C09277=1102.667,-32.003,-50.837,179.868,5.922,149.097
C09278=1102.672,-32.217,-50.825,179.868,5.919,149.097
C09279=1102.676,-32.431,-50.814,179.868,5.915,149.096
C09280=1102.682,-32.681,-50.801,179.867,5.910,149.095
C09281=1102.687,-32.930,-50.787,179.867,5.906,149.094
C09282=1102.692,-33.180,-50.774,179.867,5.902,149.093
C09283=1102.697,-33.429,-50.761,179.866,5.897,149.092
C09284=1102.702,-33.679,-50.748,179.866,5.893,149.091
C09285=1102.707,-33.928,-50.734,179.866,5.889,149.090
C09286=1102.712,-34.178,-50.721,179.865,5.884,149.089
C09287=1102.717,-34.428,-50.708,179.865,5.879,149.089
C09288=1102.723,-34.677,-50.696,179.865,5.875,149.088
C09289=1102.727,-34.927,-50.683,179.865,5.870,149.087
C09290=1102.733,-35.176,-50.669,179.864,5.866,149.086
C09291=1102.737,-35.426,-50.656,179.864,5.862,149.085
C09292=1102.743,-35.676,-50.643,179.864,5.857,149.084
C09293=1102.748,-35.926,-50.630,179.863,5.852,149.083
C09294=1102.753,-36.175,-50.617,179.864,5.848,149.082
C09295=1102.758,-36.424,-50.603,179.863,5.844,149.081
C09296=1102.763,-36.674,-50.590,179.863,5.839,149.080
C09297=1102.768,-36.924,-50.577,179.863,5.835,149.079
C09298=1102.774,-37.173,-50.564,179.862,5.830,149.079
C09299=1102.778,-37.423,-50.551,179.862,5.826,149.078
C09300=1102.783,-37.673,-50.539,179.862,5.822,149.077
C09301=1102.789,-37.923,-50.525,179.862,5.817,149.076
C09302=1102.794,-38.172,-50.513,179.861,5.812,149.075
C09303=1102.799,-38.421,-50.499,179.861,5.807,149.074
C09304=1102.804,-38.671,-50.486,179.861,5.803,149.073
C09305=1102.809,-38.921,-50.473,179.861,5.798,149.072
C09306=1102.814,-39.170,-50.460,179.860,5.794,149.071
C09307=1102.819,-39.420,-50.447,179.861,5.790,149.070
C09308=1102.825,-39.670,-50.434,179.860,5.785,149.069
C09309=1102.830,-39.919,-50.422,179.860,5.780,149.068
C09310=1102.834,-40.169,-50.409,179.860,5.775,149.067
C09311=1102.840,-40.419,-50.396,179.860,5.771,149.066
C09312=1102.845,-40.668,-50.383,179.860,5.766,149.065
C09313=1102.850,-40.918,-50.370,179.860,5.761,149.064
C09314=1102.855,-41.167,-50.357,179.860,5.757,149.063
C09315=1102.861,-41.417,-50.344,179.860,5.752,149.062
C09316=1102.865,-41.667,-50.331,179.859,5.748,149.061
C09317=1102.870,-41.916,-50.319,179.859,5.742,149.060
C09318=1102.875,-42.166,-50.306,179.859,5.738,149.059
C09319=1102.881,-42.415,-50.293,179.860,5.733,149.058
C09320=1102.886,-42.665,-50.280,179.859,5.729,149.057
C09321=1102.891,-42.915,-50.267,179.859,5.723,149.056
C09322=1102.896,-43.164,-50.255,179.860,5.719,149.055
C09323=1102.901,-43.414,-50.242,179.860,5.714,149.054
C09324=1102.906,-43.663,-50.228,179.859,5.709,149.053
C09325=1102.912,-43.913,-50.217,179.860,5.705,149.052
C09326=1102.916,-44.163,-50.204,179.860,5.700,149.050
C09327=1102.922,-44.413,-50.191,179.860,5.695,149.049
C09328=1102.926,-44.627,-50.180,179.860,5.691,149.048
C09329=1102.931,-44.841,-50.169,179.861,5.687,149.047
C09330=1102.935,-45.055,-50.159,179.861,5.683,149.046
C09331=1102.939,-45.269,-50.147,179.861,5.679,149.046
C09332=1102.943,-45.483,-50.136,179.861,5.675,149.045
C09333=1102.947,-45.697,-50.125,179.861,5.671,149.044
C09334=1102.952,-45.911,-50.115,179.861,5.667,149.043
C09335=1102.957,-46.126,-50.103,179.862,5.663,149.042
C09336=1102.962,-46.375,-50.091,179.862,5.658,149.041
C09337=1102.967,-46.626,-50.079,179.862,5.653,149.040
C09338=1102.972,-46.875,-50.066,179.862,5.649,149.039
C09339=1102.977,-47.124,-50.053,179.862,5.644,149.037
C09340=1102.982,-47.373,-50.041,179.862,5.639,149.036
C09341=1102.987,-47.623,-50.028,179.862,5.635,149.035
C09342=1102.993,-47.874,-50.015,179.862,5.630,149.034
C09343=1102.998,-48.123,-50.003,179.862,5.625,149.033
C09344=1103.003,-48.372,-49.990,179.863,5.621,149.032
C09345=1103.008,-48.622,-49.978,179.863,5.616,149.031
C09346=1103.013,-48.872,-49.965,179.863,5.610,149.030
C09347=1103.018,-49.122,-49.953,179.863,5.606,149.029
C09348=1103.023,-49.371,-49.940,179.863,5.601,149.028
C09349=1103.028,-49.620,-49.928,179.863,5.596,149.027
C09350=1103.034,-49.870,-49.916,179.864,5.592,149.026
C09351=1103.039,-50.120,-49.903,179.863,5.587,149.025
C09352=1103.044,-50.370,-49.890,179.864,5.583,149.023
C09353=1103.049,-50.619,-49.877,179.864,5.578,149.022
C09354=1103.054,-50.869,-49.866,179.864,5.573,149.021
C09355=1103.059,-51.118,-49.853,179.864,5.569,149.020
C09356=1103.064,-51.367,-49.840,179.864,5.564,149.019
C09357=1103.070,-51.617,-49.829,179.864,5.559,149.018
C09358=1103.074,-51.867,-49.816,179.865,5.555,149.017
C09359=1103.079,-52.117,-49.803,179.865,5.549,149.016
C09360=1103.085,-52.367,-49.791,179.864,5.545,149.015
C09361=1103.090,-52.616,-49.778,179.865,5.540,149.014
C09362=1103.095,-52.865,-49.766,179.865,5.535,149.013
C09363=1103.101,-53.115,-49.754,179.865,5.530,149.012
C09364=1103.105,-53.365,-49.741,179.865,5.526,149.011
C09365=1103.110,-53.615,-49.729,179.865,5.521,149.009
C09366=1103.116,-53.864,-49.717,179.865,5.516,149.008
C09367=1103.121,-54.114,-49.704,179.866,5.512,149.007
C09368=1103.126,-54.364,-49.692,179.865,5.507,149.006
C09369=1103.131,-54.613,-49.679,179.865,5.502,149.005
C09370=1103.137,-54.863,-49.668,179.866,5.498,149.004
C09371=1103.142,-55.112,-49.655,179.866,5.493,149.003
C09372=1103.146,-55.362,-49.642,179.866,5.488,149.002
C09373=1103.152,-55.612,-49.630,179.866,5.484,149.001
C09374=1103.157,-55.862,-49.617,179.866,5.479,149.000
C09375=1103.162,-56.112,-49.606,179.866,5.474,148.999
C09376=1103.167,-56.361,-49.593,179.866,5.470,148.998
C09377=1103.172,-56.610,-49.582,179.866,5.465,148.997
C09378=1103.177,-56.860,-49.569,179.866,5.460,148.995
C09379=1103.183,-57.110,-49.557,179.867,5.456,148.995
C09380=1103.188,-57.359,-49.545,179.867,5.450,148.993
C09381=1103.193,-57.609,-49.533,179.866,5.446,148.992
C09382=1103.198,-57.859,-49.520,179.867,5.441,148.991
C09383=1103.203,-58.109,-49.508,179.867,5.436,148.990
C09384=1103.208,-58.322,-49.498,179.867,5.432,148.989
C09385=1103.212,-58.537,-49.487,179.867,5.429,148.989
C09386=1103.216,-58.752,-49.477,179.867,5.424,148.988
C09387=1103.221,-58.965,-49.466,179.867,5.420,148.987
C09388=1103.225,-59.179,-49.456,179.867,5.416,148.986
C09389=1103.229,-59.394,-49.446,179.867,5.412,148.985
C09390=1103.234,-59.608,-49.435,179.867,5.408,148.984
C09391=1103.238,-59.822,-49.425,179.868,5.404,148.983
C09392=1103.243,-60.072,-49.413,179.867,5.400,148.982
C09393=1103.249,-60.322,-49.401,179.867,5.394,148.981
C09394=1103.254,-60.571,-49.388,179.867,5.390,148.980
C09395=1103.259,-60.821,-49.376,179.867,5.385,148.979
C09396=1103.264,-61.070,-49.364,179.867,5.380,148.978
C09397=1103.269,-61.320,-49.353,179.866,5.375,148.977
C09398=1103.275,-61.570,-49.341,179.866,5.370,148.976
C09399=1103.280,-61.819,-49.328,179.866,5.365,148.975
C09400=1103.284,-62.069,-49.317,179.866,5.360,148.974
C09401=1103.290,-62.319,-49.305,179.866,5.355,148.973
C09402=1103.295,-62.568,-49.292,179.866,5.350,148.972
C09403=1103.300,-62.818,-49.280,179.866,5.345,148.970
C09404=1103.305,-63.068,-49.269,179.866,5.340,148.969
C09405=1103.310,-63.317,-49.256,179.866,5.335,148.968
C09406=1103.316,-63.567,-49.245,179.865,5.330,148.967
C09407=1103.321,-63.817,-49.233,179.865,5.325,148.966
C09408=1103.326,-64.067,-49.221,179.865,5.321,148.965
C09409=1103.331,-64.316,-49.209,179.865,5.315,148.964
C09410=1103.336,-64.566,-49.197,179.865,5.310,148.963
C09411=1103.341,-64.815,-49.186,179.865,5.306,148.962
C09412=1103.346,-65.065,-49.174,179.865,5.300,148.961
C09413=1103.351,-65.315,-49.161,179.865,5.295,148.960
C09414=1103.357,-65.565,-49.149,179.865,5.291,148.959
C09415=1103.362,-65.814,-49.138,179.865,5.285,148.958
C09416=1103.367,-66.064,-49.126,179.865,5.280,148.956
C09417=1103.372,-66.314,-49.113,179.865,5.276,148.956
C09418=1103.377,-66.563,-49.102,179.865,5.270,148.954
C09419=1103.382,-66.813,-49.090,179.865,5.265,148.953
C09420=1103.388,-67.062,-49.079,179.864,5.261,148.952
C09421=1103.393,-67.312,-49.068,179.865,5.255,148.951
C09422=1103.398,-67.562,-49.056,179.865,5.250,148.950
C09423=1103.403,-67.811,-49.044,179.865,5.245,148.949
C09424=1103.408,-68.061,-49.032,179.865,5.240,148.948
C09425=1103.414,-68.311,-49.020,179.865,5.235,148.947
C09426=1103.418,-68.560,-49.009,179.865,5.230,148.945
C09427=1103.424,-68.810,-48.997,179.865,5.225,148.944
C09428=1103.429,-69.060,-48.985,179.865,5.220,148.943
C09429=1103.434,-69.310,-48.973,179.865,5.215,148.942
C09430=1103.440,-69.559,-48.962,179.865,5.210,148.941
C09431=1103.445,-69.809,-48.951,179.865,5.205,148.940
C09432=1103.450,-70.059,-48.939,179.865,5.200,148.939
C09433=1103.455,-70.308,-48.928,179.865,5.195,148.938
C09434=1103.460,-70.558,-48.916,179.865,5.189,148.936
C09435=1103.465,-70.808,-48.903,179.865,5.184,148.935
C09436=1103.470,-71.057,-48.892,179.866,5.179,148.934
C09437=1103.476,-71.306,-48.880,179.866,5.174,148.933
C09438=1103.481,-71.556,-48.869,179.865,5.169,148.932
C09439=1103.486,-71.806,-48.857,179.865,5.164,148.931
C09440=1103.490,-72.021,-48.847,179.866,5.160,148.930
C09441=1103.495,-72.235,-48.837,179.866,5.156,148.929
C09442=1103.499,-72.450,-48.828,179.866,5.151,148.928
C09443=1103.504,-72.663,-48.818,179.866,5.147,148.927
C09444=1103.508,-72.878,-48.808,179.866,5.142,148.926
C09445=1103.513,-73.092,-48.798,179.867,5.138,148.925
C09446=1103.517,-73.307,-48.788,179.867,5.134,148.924
C09447=1103.522,-73.521,-48.778,179.867,5.129,148.923
C09448=1103.527,-73.771,-48.767,179.867,5.124,148.922
C09449=1103.532,-74.021,-48.755,179.867,5.119,148.920
C09450=1103.538,-74.270,-48.744,179.867,5.114,148.919
C09451=1103.542,-74.519,-48.733,179.867,5.109,148.918
C09452=1103.548,-74.769,-48.721,179.867,5.104,148.917
C09453=1103.552,-75.019,-48.710,179.867,5.099,148.916
C09454=1103.558,-75.269,-48.698,179.868,5.093,148.915
C09455=1103.563,-75.518,-48.687,179.868,5.088,148.913
C09456=1103.569,-75.768,-48.675,179.868,5.083,148.912
C09457=1103.574,-76.018,-48.665,179.868,5.078,148.911
C09458=1103.579,-76.268,-48.653,179.868,5.073,148.910
C09459=1103.584,-76.517,-48.642,179.868,5.068,148.909
C09460=1103.590,-76.767,-48.630,179.868,5.063,148.908
C09461=1103.594,-77.016,-48.619,179.869,5.058,148.906
C09462=1103.599,-77.266,-48.607,179.869,5.053,148.905
C09463=1103.605,-77.516,-48.596,179.869,5.048,148.904
C09464=1103.610,-77.765,-48.585,179.870,5.043,148.903
C09465=1103.616,-78.015,-48.573,179.870,5.037,148.901
C09466=1103.620,-78.265,-48.562,179.870,5.032,148.900
C09467=1103.626,-78.514,-48.551,179.871,5.027,148.899
C09468=1103.631,-78.764,-48.540,179.871,5.022,148.898
C09469=1103.636,-79.014,-48.529,179.871,5.017,148.897
C09470=1103.641,-79.264,-48.517,179.871,5.012,148.896
C09471=1103.647,-79.513,-48.506,179.871,5.007,148.894
C09472=1103.652,-79.763,-48.495,179.871,5.001,148.893
C09473=1103.657,-80.013,-48.483,179.872,4.996,148.892
C09474=1103.662,-80.262,-48.472,179.872,4.991,148.891
C09475=1103.667,-80.512,-48.462,179.872,4.986,148.890
C09476=1103.673,-80.762,-48.450,179.872,4.981,148.888
C09477=1103.678,-81.011,-48.439,179.872,4.976,148.887
C09478=1103.683,-81.261,-48.428,179.873,4.971,148.886
C09479=1103.689,-81.511,-48.417,179.874,4.966,148.885
C09480=1103.693,-81.761,-48.405,179.874,4.961,148.883
C09481=1103.699,-82.010,-48.394,179.874,4.956,148.882
C09482=1103.704,-82.260,-48.384,179.874,4.950,148.881
C09483=1103.709,-82.510,-48.372,179.874,4.945,148.880
C09484=1103.714,-82.759,-48.361,179.874,4.940,148.879
C09485=1103.719,-83.009,-48.350,179.875,4.935,148.878
C09486=1103.725,-83.259,-48.338,179.875,4.930,148.876
C09487=1103.730,-83.509,-48.328,179.875,4.925,148.875
C09488=1103.735,-83.758,-48.317,179.876,4.919,148.874
C09489=1103.740,-84.008,-48.306,179.876,4.915,148.873
C09490=1103.746,-84.258,-48.295,179.877,4.910,148.871
C09491=1103.751,-84.507,-48.284,179.877,4.905,148.870
C09492=1103.756,-84.757,-48.273,179.877,4.899,148.869
C09493=1103.761,-85.007,-48.262,179.877,4.894,148.868
C09494=1103.766,-85.256,-48.251,179.877,4.889,148.867
C09495=1103.772,-85.506,-48.240,179.877,4.884,148.866
C09496=1103.776,-85.721,-48.231,179.878,4.880,148.864
C09497=1103.781,-85.935,-48.221,179.879,4.876,148.863
C09498=1103.785,-86.149,-48.212,179.878,4.871,148.862
C09499=1103.789,-86.364,-48.203,179.879,4.867,148.861
C09500=1103.794,-86.578,-48.193,179.879,4.863,148.860
C09501=1103.798,-86.793,-48.184,179.880,4.858,148.859
C09502=1103.803,-87.007,-48.174,179.880,4.854,148.858
C09503=1103.807,-87.221,-48.165,179.880,4.850,148.857
C09504=1103.812,-87.471,-48.154,179.880,4.845,148.856
C09505=1103.818,-87.720,-48.143,179.881,4.839,148.855
C09506=1103.823,-87.970,-48.132,179.881,4.834,148.853
C09507=1103.828,-88.220,-48.121,179.882,4.830,148.852
C09508=1103.833,-88.470,-48.111,179.882,4.824,148.851
C09509=1103.838,-88.719,-48.099,179.882,4.819,148.850
C09510=1103.844,-88.969,-48.089,179.882,4.814,148.849
C09511=1103.849,-89.219,-48.079,179.883,4.809,148.847
C09512=1103.854,-89.469,-48.067,179.883,4.805,148.846
C09513=1103.860,-89.719,-48.057,179.883,4.799,148.845
C09514=1103.864,-89.968,-48.045,179.884,4.794,148.844
C09515=1103.870,-90.218,-48.035,179.884,4.789,148.843
C09516=1103.875,-90.467,-48.024,179.885,4.785,148.842
C09517=1103.880,-90.717,-48.014,179.885,4.780,148.840
C09518=1103.885,-90.967,-48.003,179.886,4.774,148.839
C09519=1103.891,-91.216,-47.992,179.886,4.769,148.838
C09520=1103.896,-91.466,-47.981,179.886,4.764,148.837
C09521=1103.901,-91.717,-47.971,179.887,4.760,148.835
C09522=1103.907,-91.966,-47.959,179.887,4.754,148.834
C09523=1103.912,-92.216,-47.949,179.887,4.749,148.833
C09524=1103.917,-92.465,-47.938,179.888,4.745,148.832
C09525=1103.922,-92.715,-47.927,179.888,4.740,148.831
C09526=1103.928,-92.965,-47.917,179.888,4.735,148.829
C09527=1103.932,-93.214,-47.906,179.888,4.729,148.828
C09528=1103.938,-93.464,-47.896,179.889,4.725,148.827
C09529=1103.943,-93.714,-47.885,179.889,4.720,148.826
C09530=1103.948,-93.964,-47.875,179.890,4.715,148.825
C09531=1103.953,-94.213,-47.864,179.890,4.711,148.823
C09532=1103.959,-94.463,-47.853,179.891,4.705,148.822
C09533=1103.964,-94.713,-47.843,179.891,4.700,148.821
C09534=1103.969,-94.962,-47.832,179.892,4.696,148.820
C09535=1103.974,-95.212,-47.821,179.892,4.691,148.819
C09536=1103.980,-95.462,-47.811,179.892,4.686,148.817
C09537=1103.985,-95.712,-47.800,179.892,4.680,148.816
C09538=1103.990,-95.961,-47.790,179.893,4.676,148.815
C09539=1103.995,-96.211,-47.779,179.893,4.671,148.814
C09540=1104.000,-96.461,-47.769,179.893,4.666,148.813
C09541=1104.005,-96.711,-47.758,179.894,4.662,148.812
C09542=1104.011,-96.960,-47.747,179.894,4.656,148.810
C09543=1104.016,-97.209,-47.737,179.895,4.651,148.809
C09544=1104.021,-97.460,-47.726,179.895,4.647,148.808
C09545=1104.027,-97.709,-47.716,179.896,4.642,148.807
C09546=1104.032,-97.960,-47.706,179.896,4.637,148.806
C09547=1104.038,-98.209,-47.695,179.897,4.632,148.804
C09548=1104.042,-98.459,-47.684,179.897,4.627,148.803
C09549=1104.048,-98.708,-47.674,179.897,4.622,148.802
C09550=1104.053,-98.958,-47.664,179.898,4.618,148.801
C09551=1104.058,-99.208,-47.654,179.898,4.612,148.800
C09552=1104.063,-99.422,-47.644,179.898,4.609,148.799
C09553=1104.067,-99.636,-47.636,179.899,4.603,148.797
C09554=1104.072,-99.852,-47.627,179.899,4.599,148.796
C09555=1104.076,-100.066,-47.618,179.899,4.595,148.795
C09556=1104.080,-100.280,-47.609,179.900,4.591,148.794
C09557=1104.085,-100.494,-47.600,179.900,4.587,148.793
C09558=1104.090,-100.709,-47.591,179.901,4.583,148.792
C09559=1104.094,-100.924,-47.583,179.901,4.578,148.791
C09560=1104.099,-101.173,-47.572,179.902,4.574,148.790
C09561=1104.105,-101.422,-47.561,179.902,4.569,148.789
C09562=1104.110,-101.673,-47.551,179.902,4.563,148.788
C09563=1104.115,-101.922,-47.541,179.903,4.559,148.786
C09564=1104.120,-102.172,-47.530,179.903,4.554,148.785
C09565=1104.126,-102.422,-47.520,179.903,4.549,148.784
C09566=1104.131,-102.671,-47.510,179.904,4.544,148.783
C09567=1104.136,-102.921,-47.500,179.904,4.539,148.782
C09568=1104.141,-103.171,-47.489,179.905,4.534,148.780
C09569=1104.146,-103.421,-47.479,179.905,4.529,148.779
C09570=1104.152,-103.671,-47.469,179.906,4.525,148.778
C09571=1104.158,-103.920,-47.458,179.906,4.520,148.777
C09572=1104.162,-104.170,-47.448,179.907,4.514,148.775
C09573=1104.167,-104.420,-47.438,179.907,4.509,148.774
C09574=1104.173,-104.669,-47.428,179.908,4.505,148.773
C09575=1104.178,-104.920,-47.417,179.908,4.499,148.772
C09576=1104.184,-105.169,-47.407,179.908,4.494,148.771
C09577=1104.188,-105.418,-47.398,179.908,4.489,148.769
C09578=1104.193,-105.669,-47.387,179.909,4.485,148.768
C09579=1104.199,-105.918,-47.377,179.910,4.480,148.767
C09580=1104.205,-106.168,-47.367,179.910,4.474,148.766
C09581=1104.209,-106.418,-47.357,179.910,4.469,148.764
C09582=1104.215,-106.667,-47.346,179.911,4.465,148.763
C09583=1104.220,-106.917,-47.336,179.912,4.459,148.762
C09584=1104.225,-107.167,-47.326,179.912,4.454,148.761
C09585=1104.230,-107.416,-47.316,179.912,4.449,148.759
C09586=1104.236,-107.666,-47.307,179.913,4.445,148.758
C09587=1104.241,-107.917,-47.296,179.913,4.440,148.757
C09588=1104.246,-108.166,-47.286,179.913,4.434,148.756
C09589=1104.251,-108.415,-47.276,179.914,4.429,148.755
C09590=1104.256,-108.666,-47.266,179.914,4.425,148.753
C09591=1104.262,-108.915,-47.255,179.915,4.419,148.752
C09592=1104.268,-109.165,-47.245,179.915,4.414,148.751
C09593=1104.272,-109.414,-47.236,179.916,4.409,148.750
C09594=1104.278,-109.665,-47.226,179.917,4.405,148.748
C09595=1104.283,-109.914,-47.215,179.917,4.400,148.747
C09596=1104.288,-110.164,-47.206,179.917,4.395,148.746
C09597=1104.293,-110.414,-47.195,179.917,4.389,148.745
C09598=1104.299,-110.663,-47.185,179.918,4.384,148.743
C09599=1104.304,-110.913,-47.176,179.919,4.379,148.742
C09600=1104.310,-111.163,-47.166,179.919,4.374,148.741
C09601=1104.315,-111.413,-47.155,179.919,4.369,148.740
C09602=1104.319,-111.662,-47.146,179.920,4.364,148.738
C09603=1104.325,-111.912,-47.136,179.921,4.359,148.737
C09604=1104.331,-112.162,-47.126,179.921,4.354,148.736
C09605=1104.335,-112.412,-47.116,179.921,4.349,148.735
C09606=1104.341,-112.661,-47.106,179.922,4.344,148.733
C09607=1104.346,-112.911,-47.096,179.922,4.339,148.732
C09608=1104.351,-113.125,-47.087,179.923,4.334,148.731
C09609=1104.355,-113.340,-47.079,179.923,4.330,148.730
C09610=1104.360,-113.554,-47.071,179.924,4.326,148.729
C09611=1104.364,-113.769,-47.062,179.924,4.321,148.728
C09612=1104.368,-113.984,-47.054,179.925,4.317,148.727
C09613=1104.373,-114.198,-47.045,179.925,4.313,148.726
C09614=1104.377,-114.413,-47.037,179.925,4.308,148.724
C09615=1104.383,-114.628,-47.028,179.926,4.304,148.723
C09616=1104.387,-114.877,-47.019,179.926,4.299,148.722
C09617=1104.393,-115.127,-47.009,179.927,4.293,148.721
C09618=1104.398,-115.376,-46.999,179.927,4.289,148.720
C09619=1104.403,-115.627,-46.989,179.928,4.284,148.718
C09620=1104.409,-115.877,-46.979,179.928,4.279,148.717
C09621=1104.414,-116.126,-46.970,179.929,4.273,148.716
C09622=1104.420,-116.375,-46.960,179.929,4.268,148.714
C09623=1104.425,-116.625,-46.951,179.929,4.263,148.713
C09624=1104.430,-116.876,-46.940,179.931,4.258,148.712
C09625=1104.435,-117.125,-46.930,179.931,4.253,148.711
C09626=1104.440,-117.375,-46.921,179.931,4.248,148.709
C09627=1104.445,-117.624,-46.911,179.931,4.243,148.708
C09628=1104.451,-117.874,-46.902,179.932,4.237,148.707
C09629=1104.456,-118.124,-46.892,179.933,4.232,148.705
C09630=1104.462,-118.373,-46.882,179.933,4.227,148.704
C09631=1104.467,-118.624,-46.872,179.934,4.222,148.703
C09632=1104.472,-118.873,-46.863,179.934,4.217,148.702
C09633=1104.478,-119.123,-46.853,179.935,4.212,148.700
C09634=1104.483,-119.373,-46.843,179.936,4.206,148.699
C09635=1104.489,-119.623,-46.834,179.936,4.201,148.698
C09636=1104.493,-119.872,-46.824,179.936,4.196,148.696
C09637=1104.499,-120.122,-46.815,179.937,4.190,148.695
C09638=1104.504,-120.372,-46.805,179.937,4.185,148.694
C09639=1104.509,-120.622,-46.796,179.939,4.180,148.692
C09640=1104.514,-120.872,-46.786,179.939,4.175,148.691
C09641=1104.519,-121.121,-46.777,179.939,4.170,148.690
C09642=1104.525,-121.371,-46.767,179.940,4.165,148.688
C09643=1104.530,-121.621,-46.758,179.940,4.159,148.687
C09644=1104.536,-121.870,-46.748,179.940,4.154,148.686
C09645=1104.541,-122.120,-46.739,179.941,4.149,148.684
C09646=1104.547,-122.370,-46.728,179.942,4.144,148.683
C09647=1104.551,-122.620,-46.719,179.942,4.138,148.682
C09648=1104.556,-122.870,-46.710,179.943,4.133,148.681
C09649=1104.562,-123.120,-46.700,179.943,4.127,148.679
C09650=1104.567,-123.369,-46.690,179.944,4.123,148.678
C09651=1104.573,-123.619,-46.681,179.945,4.118,148.677
C09652=1104.578,-123.868,-46.671,179.945,4.112,148.675
C09653=1104.583,-124.118,-46.662,179.946,4.107,148.674
C09654=1104.589,-124.368,-46.653,179.947,4.102,148.673
C09655=1104.593,-124.618,-46.643,179.947,4.096,148.671
C09656=1104.599,-124.868,-46.634,179.948,4.091,148.670
C09657=1104.604,-125.117,-46.624,179.948,4.086,148.669
C09658=1104.609,-125.367,-46.615,179.949,4.080,148.667
C09659=1104.615,-125.617,-46.606,179.949,4.075,148.666
C09660=1104.620,-125.866,-46.596,179.950,4.070,148.664
C09661=1104.625,-126.116,-46.587,179.950,4.064,148.663
C09662=1104.631,-126.366,-46.578,179.951,4.059,148.662
C09663=1104.635,-126.616,-46.568,179.951,4.054,148.661
C09664=1104.640,-126.831,-46.560,179.952,4.049,148.659
C09665=1104.645,-127.045,-46.552,179.952,4.044,148.658
C09666=1104.650,-127.259,-46.544,179.953,4.040,148.657
C09667=1104.655,-127.475,-46.536,179.953,4.035,148.656
C09668=1104.659,-127.689,-46.529,179.954,4.031,148.655
C09669=1104.663,-127.903,-46.520,179.955,4.026,148.653
C09670=1104.668,-128.118,-46.513,179.955,4.021,148.652
C09671=1104.672,-128.333,-46.504,179.956,4.017,148.651
C09672=1104.250,-128.323,-46.531,179.963,4.021,148.650
C09673=1104.244,-128.109,-46.538,179.962,4.026,148.651
C09674=1104.240,-127.895,-46.546,179.962,4.030,148.652
C09675=1104.235,-127.680,-46.555,179.962,4.035,148.653
C09676=1104.230,-127.465,-46.562,179.961,4.039,148.654
C09677=1104.227,-127.251,-46.570,179.961,4.044,148.656
C09678=1104.222,-127.036,-46.578,179.960,4.049,148.657
C09679=1104.217,-126.821,-46.586,179.959,4.053,148.658
C09680=1104.213,-126.607,-46.594,179.959,4.058,148.659
C09681=1104.207,-126.357,-46.604,179.958,4.063,148.661
C09682=1104.202,-126.107,-46.613,179.958,4.069,148.662
C09683=1104.197,-125.858,-46.622,179.957,4.074,148.663
C09684=1104.191,-125.608,-46.632,179.957,4.079,148.664
C09685=1104.187,-125.358,-46.642,179.956,4.085,148.666
C09686=1104.182,-125.108,-46.651,179.956,4.090,148.667
C09687=1104.176,-124.858,-46.661,179.955,4.096,148.669
C09688=1104.171,-124.608,-46.670,179.954,4.100,148.670
C09689=1104.165,-124.359,-46.680,179.953,4.105,148.671
C09690=1104.160,-124.109,-46.689,179.953,4.111,148.673
C09691=1104.155,-123.859,-46.698,179.952,4.116,148.674
C09692=1104.149,-123.610,-46.708,179.952,4.121,148.675
C09693=1104.144,-123.360,-46.717,179.951,4.127,148.677
C09694=1104.139,-123.110,-46.727,179.951,4.132,148.678
C09695=1104.133,-122.860,-46.736,179.950,4.138,148.679
C09696=1104.128,-122.611,-46.746,179.950,4.143,148.681
C09697=1104.123,-122.360,-46.755,179.949,4.148,148.682
C09698=1104.118,-122.111,-46.765,179.948,4.153,148.683
C09699=1104.112,-121.861,-46.774,179.948,4.159,148.684
C09700=1104.108,-121.612,-46.784,179.947,4.163,148.686
C09701=1104.102,-121.361,-46.794,179.947,4.168,148.687
C09702=1104.097,-121.112,-46.803,179.946,4.174,148.688
C09703=1104.091,-120.862,-46.813,179.945,4.179,148.690
C09704=1104.086,-120.613,-46.822,179.945,4.184,148.691
C09705=1104.081,-120.362,-46.832,179.944,4.190,148.693
C09706=1104.076,-120.113,-46.842,179.944,4.195,148.694
C09707=1104.070,-119.863,-46.852,179.944,4.200,148.695
C09708=1104.065,-119.613,-46.861,179.943,4.206,148.696
C09709=1104.060,-119.364,-46.871,179.942,4.210,148.698
C09710=1104.054,-119.114,-46.880,179.942,4.215,148.699
C09711=1104.049,-118.864,-46.890,179.941,4.221,148.700
C09712=1104.044,-118.614,-46.899,179.941,4.226,148.702
C09713=1104.039,-118.364,-46.910,179.940,4.231,148.703
C09714=1104.034,-118.115,-46.919,179.940,4.236,148.704
C09715=1104.028,-117.865,-46.929,179.939,4.242,148.705
C09716=1104.023,-117.616,-46.938,179.939,4.246,148.707
C09717=1104.017,-117.366,-46.949,179.938,4.252,148.708
C09718=1104.012,-117.115,-46.958,179.938,4.257,148.709
C09719=1104.007,-116.866,-46.968,179.937,4.262,148.711
C09720=1104.002,-116.616,-46.978,179.936,4.267,148.712
C09721=1103.996,-116.367,-46.987,179.936,4.273,148.713
C09722=1103.991,-116.117,-46.997,179.935,4.277,148.714
C09723=1103.987,-115.867,-47.007,179.935,4.282,148.716
C09724=1103.981,-115.617,-47.017,179.934,4.288,148.717
C09725=1103.975,-115.367,-47.027,179.934,4.293,148.718
C09726=1103.970,-115.118,-47.037,179.934,4.298,148.720
C09727=1103.964,-114.868,-47.046,179.933,4.303,148.721
C09728=1103.960,-114.618,-47.056,179.932,4.308,148.722
C09729=1103.955,-114.403,-47.065,179.932,4.312,148.723
C09730=1103.950,-114.189,-47.073,179.932,4.317,148.724
C09731=1103.946,-113.974,-47.082,179.931,4.321,148.725
C09732=1103.941,-113.760,-47.090,179.930,4.325,148.727
C09733=1103.937,-113.545,-47.098,179.931,4.330,148.728
C09734=1103.932,-113.331,-47.107,179.930,4.334,148.729
C09735=1103.928,-113.117,-47.116,179.929,4.338,148.730
C09736=1103.923,-112.902,-47.125,179.929,4.343,148.731
C09737=1103.918,-112.652,-47.134,179.928,4.348,148.732
C09738=1103.913,-112.402,-47.144,179.928,4.353,148.733
C09739=1103.907,-112.153,-47.154,179.928,4.358,148.735
C09740=1103.902,-111.903,-47.164,179.928,4.363,148.736
C09741=1103.897,-111.653,-47.175,179.926,4.368,148.737
C09742=1103.891,-111.403,-47.184,179.926,4.373,148.738
C09743=1103.886,-111.154,-47.194,179.926,4.378,148.740
C09744=1103.881,-110.904,-47.204,179.925,4.383,148.741
C09745=1103.876,-110.654,-47.214,179.925,4.388,148.742
C09746=1103.871,-110.405,-47.224,179.924,4.393,148.743
C09747=1103.865,-110.155,-47.234,179.924,4.398,148.745
C09748=1103.860,-109.904,-47.244,179.923,4.403,148.746
C09749=1103.855,-109.655,-47.254,179.923,4.409,148.747
C09750=1103.850,-109.406,-47.264,179.922,4.413,148.748
C09751=1103.844,-109.156,-47.274,179.922,4.418,148.750
C09752=1103.839,-108.906,-47.285,179.922,4.423,148.751
C09753=1103.834,-108.657,-47.294,179.921,4.429,148.752
C09754=1103.829,-108.407,-47.305,179.921,4.434,148.753
C09755=1103.824,-108.157,-47.315,179.920,4.438,148.755
C09756=1103.818,-107.907,-47.325,179.920,4.443,148.756
C09757=1103.813,-107.657,-47.334,179.919,4.449,148.757
C09758=1103.808,-107.407,-47.345,179.919,4.454,148.758
C09759=1103.802,-107.158,-47.355,179.918,4.458,148.759
C09760=1103.797,-106.908,-47.365,179.918,4.463,148.761
C09761=1103.792,-106.658,-47.375,179.917,4.469,148.762
C09762=1103.787,-106.409,-47.385,179.917,4.473,148.763
C09763=1103.781,-106.159,-47.396,179.916,4.478,148.764
C09764=1103.776,-105.909,-47.406,179.916,4.483,148.766
C09765=1103.771,-105.659,-47.416,179.916,4.489,148.767
C09766=1103.766,-105.410,-47.426,179.915,4.493,148.768
C09767=1103.761,-105.160,-47.437,179.915,4.498,148.769
C09768=1103.755,-104.910,-47.447,179.915,4.503,148.770
C09769=1103.749,-104.661,-47.457,179.914,4.508,148.772
C09770=1103.744,-104.410,-47.468,179.914,4.513,148.773
C09771=1103.740,-104.161,-47.477,179.913,4.518,148.774
C09772=1103.735,-103.911,-47.488,179.913,4.523,148.776
C09773=1103.729,-103.661,-47.498,179.912,4.528,148.777
C09774=1103.723,-103.412,-47.508,179.912,4.533,148.778
C09775=1103.718,-103.162,-47.519,179.911,4.538,148.779
C09776=1103.713,-102.912,-47.529,179.911,4.543,148.780
C09777=1103.709,-102.662,-47.539,179.910,4.547,148.782
C09778=1103.703,-102.413,-47.549,179.910,4.553,148.783
C09779=1103.698,-102.164,-47.560,179.910,4.558,148.784
C09780=1103.693,-101.913,-47.571,179.910,4.563,148.785
C09781=1103.687,-101.664,-47.581,179.909,4.567,148.786
C09782=1103.682,-101.414,-47.591,179.909,4.572,148.788
C09783=1103.677,-101.164,-47.602,179.908,4.578,148.789
C09784=1103.671,-100.915,-47.612,179.908,4.582,148.790
C09785=1103.667,-100.700,-47.621,179.907,4.587,148.791
C09786=1103.663,-100.486,-47.630,179.907,4.591,148.792
C09787=1103.658,-100.271,-47.638,179.907,4.595,148.793
C09788=1103.653,-100.057,-47.648,179.906,4.599,148.794
C09789=1103.649,-99.842,-47.656,179.906,4.603,148.795
C09790=1103.645,-99.628,-47.666,179.905,4.607,148.796
C09791=1103.640,-99.413,-47.674,179.905,4.612,148.797
C09792=1103.635,-99.199,-47.684,179.905,4.616,148.798
C09793=1103.631,-98.949,-47.694,179.904,4.621,148.800
C09794=1103.625,-98.700,-47.704,179.904,4.626,148.801
C09795=1103.620,-98.450,-47.714,179.904,4.631,148.802
C09796=1103.615,-98.200,-47.725,179.903,4.636,148.803
C09797=1103.609,-97.951,-47.736,179.903,4.640,148.804
C09798=1103.604,-97.701,-47.746,179.902,4.646,148.806
C09799=1103.599,-97.451,-47.757,179.902,4.651,148.807
C09800=1103.594,-97.201,-47.767,179.901,4.655,148.808
C09801=1103.588,-96.952,-47.778,179.901,4.660,148.809
C09802=1103.583,-96.702,-47.789,179.901,4.665,148.810
C09803=1103.578,-96.452,-47.799,179.900,4.670,148.811
C09804=1103.573,-96.202,-47.809,179.900,4.675,148.813
C09805=1103.568,-95.953,-47.820,179.900,4.680,148.814
C09806=1103.563,-95.703,-47.831,179.899,4.684,148.815
C09807=1103.557,-95.453,-47.841,179.899,4.689,148.816
C09808=1103.552,-95.203,-47.852,179.898,4.695,148.817
C09809=1103.547,-94.954,-47.863,179.898,4.699,148.819
C09810=1103.542,-94.704,-47.873,179.897,4.704,148.820
C09811=1103.536,-94.454,-47.883,179.897,4.709,148.821
C09812=1103.531,-94.205,-47.895,179.896,4.714,148.822
C09813=1103.526,-93.955,-47.905,179.896,4.719,148.823
C09814=1103.521,-93.705,-47.915,179.896,4.724,148.825
C09815=1103.515,-93.456,-47.927,179.896,4.729,148.826
C09816=1103.510,-93.205,-47.938,179.895,4.733,148.827
C09817=1103.504,-92.956,-47.948,179.895,4.738,148.828
C09818=1103.499,-92.706,-47.959,179.895,4.744,148.829
C09819=1103.494,-92.457,-47.969,179.894,4.748,148.831
C09820=1103.489,-92.206,-47.980,179.894,4.753,148.832
C09821=1103.484,-91.957,-47.991,179.894,4.758,148.833
C09822=1103.479,-91.707,-48.001,179.893,4.763,148.834
C09823=1103.473,-91.458,-48.012,179.893,4.768,148.835
C09824=1103.468,-91.208,-48.023,179.892,4.773,148.837
C09825=1103.463,-90.958,-48.033,179.892,4.778,148.838
C09826=1103.458,-90.709,-48.044,179.891,4.783,148.839
C09827=1103.452,-90.458,-48.055,179.891,4.789,148.840
C09828=1103.447,-90.209,-48.066,179.890,4.793,148.842
C09829=1103.442,-89.959,-48.077,179.890,4.798,148.843
C09830=1103.436,-89.710,-48.087,179.890,4.803,148.844
C09831=1103.432,-89.460,-48.098,179.890,4.808,148.845
C09832=1103.427,-89.210,-48.109,179.889,4.813,148.846
C09833=1103.421,-88.961,-48.120,179.889,4.818,148.847
C09834=1103.416,-88.710,-48.131,179.889,4.823,148.849
C09835=1103.410,-88.461,-48.142,179.889,4.828,148.850
C09836=1103.405,-88.211,-48.153,179.888,4.833,148.851
C09837=1103.401,-87.961,-48.164,179.888,4.838,148.852
C09838=1103.395,-87.712,-48.174,179.887,4.843,148.854
C09839=1103.390,-87.462,-48.185,179.887,4.848,148.855
C09840=1103.384,-87.212,-48.196,179.887,4.853,148.856
C09841=1103.380,-86.998,-48.206,179.886,4.857,148.857
C09842=1103.376,-86.784,-48.215,179.887,4.862,148.858
C09843=1103.371,-86.570,-48.224,179.886,4.866,148.859
C09844=1103.367,-86.355,-48.234,179.886,4.870,148.860
C09845=1103.363,-86.141,-48.243,179.885,4.876,148.861
C09846=1103.358,-85.926,-48.253,179.885,4.880,148.862
C09847=1103.353,-85.711,-48.262,179.885,4.883,148.863
C09848=1103.349,-85.498,-48.271,179.884,4.888,148.864
C09849=1103.344,-85.248,-48.283,179.884,4.893,148.865
C09850=1103.339,-84.997,-48.294,179.884,4.898,148.867
C09851=1103.333,-84.749,-48.305,179.884,4.903,148.868
C09852=1103.329,-84.499,-48.316,179.883,4.908,148.869
C09853=1103.323,-84.249,-48.326,179.883,4.913,148.870
C09854=1103.318,-83.999,-48.338,179.883,4.919,148.871
C09855=1103.313,-83.749,-48.349,179.883,4.924,148.873
C09856=1103.307,-83.500,-48.360,179.882,4.929,148.874
C09857=1103.302,-83.250,-48.371,179.881,4.934,148.875
C09858=1103.297,-83.000,-48.382,179.881,4.939,148.876
C09859=1103.292,-82.750,-48.393,179.881,4.944,148.878
C09860=1103.287,-82.502,-48.404,179.881,4.949,148.879
C09861=1103.281,-82.251,-48.415,179.881,4.954,148.880
C09862=1103.276,-82.001,-48.427,179.881,4.959,148.881
C09863=1103.271,-81.752,-48.438,179.880,4.964,148.882
C09864=1103.265,-81.502,-48.449,179.880,4.970,148.883
C09865=1103.261,-81.252,-48.460,179.880,4.975,148.885
C09866=1103.255,-81.003,-48.471,179.879,4.980,148.886
C09867=1103.250,-80.753,-48.483,179.879,4.985,148.887
C09868=1103.245,-80.503,-48.494,179.879,4.990,148.888
C09869=1103.240,-80.253,-48.505,179.878,4.995,148.890
C09870=1103.234,-80.004,-48.516,179.878,5.000,148.891
C09871=1103.230,-79.755,-48.528,179.878,5.005,148.892
C09872=1103.225,-79.504,-48.538,179.878,5.010,148.893
C09873=1103.219,-79.255,-48.550,179.878,5.015,148.894
C09874=1103.214,-79.006,-48.561,179.878,5.021,148.895
C09875=1103.208,-78.756,-48.573,179.877,5.026,148.897
C09876=1103.204,-78.506,-48.584,179.877,5.031,148.898
C09877=1103.198,-78.256,-48.594,179.877,5.036,148.899
C09878=1103.193,-78.006,-48.606,179.876,5.041,148.900
C09879=1103.188,-77.757,-48.618,179.876,5.047,148.902
C09880=1103.183,-77.507,-48.629,179.876,5.052,148.903
C09881=1103.177,-77.258,-48.640,179.876,5.057,148.904
C09882=1103.172,-77.007,-48.652,179.876,5.062,148.905
C09883=1103.167,-76.758,-48.663,179.876,5.067,148.906
C09884=1103.162,-76.508,-48.674,179.876,5.072,148.907
C09885=1103.156,-76.259,-48.686,179.875,5.077,148.909
C09886=1103.151,-76.009,-48.697,179.875,5.082,148.910
C09887=1103.146,-75.759,-48.709,179.874,5.087,148.911
C09888=1103.141,-75.510,-48.720,179.874,5.092,148.912
C09889=1103.136,-75.260,-48.732,179.874,5.097,148.913
C09890=1103.131,-75.011,-48.743,179.874,5.102,148.915
C09891=1103.125,-74.760,-48.754,179.874,5.107,148.916
C09892=1103.120,-74.511,-48.765,179.874,5.113,148.917
C09893=1103.115,-74.261,-48.777,179.874,5.118,148.918
C09894=1103.110,-74.011,-48.789,179.873,5.123,148.919
C09895=1103.104,-73.762,-48.800,179.873,5.128,148.920
C09896=1103.099,-73.512,-48.811,179.873,5.133,148.922
C09897=1103.095,-73.297,-48.821,179.874,5.138,148.923
C09898=1103.090,-73.084,-48.832,179.873,5.142,148.923
C09899=1103.086,-72.869,-48.842,179.873,5.146,148.925
C09900=1103.081,-72.655,-48.851,179.873,5.151,148.926
C09901=1103.077,-72.440,-48.861,179.873,5.155,148.927
C09902=1103.073,-72.227,-48.871,179.873,5.160,148.927
C09903=1103.069,-72.012,-48.881,179.872,5.164,148.929
C09904=1103.064,-71.798,-48.891,179.872,5.168,148.930
C09905=1103.058,-71.548,-48.903,179.872,5.173,148.931
C09906=1103.053,-71.298,-48.914,179.872,5.178,148.932
C09907=1103.048,-71.048,-48.926,179.872,5.183,148.933
C09908=1103.043,-70.799,-48.937,179.872,5.188,148.934
C09909=1103.038,-70.550,-48.949,179.872,5.193,148.935
C09910=1103.033,-70.300,-48.961,179.872,5.198,148.936
C09911=1103.027,-70.051,-48.973,179.872,5.203,148.938
C09912=1103.022,-69.801,-48.984,179.872,5.209,148.939
C09913=1103.017,-69.551,-48.996,179.871,5.214,148.940
C09914=1103.012,-69.301,-49.008,179.871,5.219,148.941
C09915=1103.007,-69.051,-49.019,179.872,5.224,148.942
C09916=1103.002,-68.801,-49.031,179.872,5.229,148.943
C09917=1102.996,-68.551,-49.043,179.871,5.234,148.944
C09918=1102.991,-68.303,-49.054,179.871,5.239,148.945
C09919=1102.986,-68.053,-49.066,179.871,5.244,148.947
C09920=1102.981,-67.803,-49.078,179.871,5.249,148.948
C09921=1102.976,-67.554,-49.089,179.871,5.254,148.949
C09922=1102.970,-67.304,-49.101,179.871,5.259,148.950
C09923=1102.965,-67.054,-49.113,179.871,5.264,148.951
C09924=1102.960,-66.804,-49.124,179.871,5.269,148.952
C09925=1102.955,-66.555,-49.137,179.871,5.274,148.953
C09926=1102.950,-66.305,-49.149,179.871,5.279,148.954
C09927=1102.945,-66.055,-49.160,179.871,5.284,148.955
C09928=1102.940,-65.805,-49.172,179.872,5.289,148.956
C09929=1102.935,-65.556,-49.185,179.871,5.294,148.958
C09930=1102.930,-65.306,-49.196,179.871,5.299,148.959
C09931=1102.924,-65.057,-49.208,179.872,5.304,148.960
C09932=1102.919,-64.807,-49.220,179.872,5.309,148.961
C09933=1102.915,-64.558,-49.232,179.871,5.314,148.962
C09934=1102.909,-64.308,-49.244,179.872,5.319,148.963
C09935=1102.904,-64.058,-49.255,179.872,5.324,148.964
C09936=1102.898,-63.808,-49.267,179.872,5.329,148.965
C09937=1102.894,-63.559,-49.279,179.872,5.334,148.966
C09938=1102.888,-63.309,-49.291,179.872,5.339,148.967
C09939=1102.883,-63.059,-49.303,179.872,5.344,148.968
C09940=1102.878,-62.810,-49.316,179.872,5.349,148.969
C09941=1102.873,-62.560,-49.327,179.873,5.354,148.970
C09942=1102.868,-62.310,-49.339,179.872,5.359,148.972
C09943=1102.863,-62.061,-49.352,179.872,5.364,148.973
C09944=1102.857,-61.811,-49.363,179.872,5.368,148.974
C09945=1102.852,-61.561,-49.376,179.872,5.373,148.975
C09946=1102.847,-61.312,-49.387,179.872,5.378,148.976
C09947=1102.842,-61.062,-49.399,179.873,5.383,148.977
C09948=1102.837,-60.813,-49.412,179.873,5.388,148.978
C09949=1102.831,-60.563,-49.424,179.873,5.393,148.979
C09950=1102.826,-60.313,-49.436,179.873,5.398,148.980
C09951=1102.822,-60.064,-49.448,179.873,5.403,148.981
C09952=1102.816,-59.814,-49.459,179.873,5.408,148.982
C09953=1102.812,-59.599,-49.470,179.874,5.411,148.983
C09954=1102.808,-59.386,-49.481,179.873,5.415,148.984
C09955=1102.803,-59.171,-49.492,179.874,5.420,148.985
C09956=1102.798,-58.957,-49.502,179.874,5.424,148.985
C09957=1102.794,-58.743,-49.512,179.873,5.428,148.986
C09958=1102.790,-58.529,-49.523,179.873,5.432,148.987
C09959=1102.785,-58.315,-49.533,179.873,5.436,148.988
C09960=1102.781,-58.100,-49.543,179.873,5.440,148.989
C09961=1102.776,-57.851,-49.556,179.873,5.445,148.990
C09962=1102.770,-57.601,-49.568,179.873,5.449,148.991
C09963=1102.765,-57.352,-49.580,179.872,5.454,148.992
C09964=1102.760,-57.101,-49.593,179.873,5.459,148.993
C09965=1102.756,-56.852,-49.605,179.873,5.464,148.995
C09966=1102.750,-56.602,-49.617,179.872,5.468,148.995
C09967=1102.745,-56.353,-49.629,179.872,5.473,148.997
C09968=1102.740,-56.103,-49.641,179.872,5.478,148.998
C09969=1102.735,-55.854,-49.654,179.872,5.482,148.999
C09970=1102.729,-55.604,-49.665,179.872,5.487,149.000
C09971=1102.724,-55.354,-49.678,179.872,5.492,149.001
C09972=1102.719,-55.105,-49.691,179.872,5.496,149.002
C09973=1102.714,-54.854,-49.703,179.872,5.501,149.003
C09974=1102.709,-54.605,-49.716,179.872,5.506,149.004
C09975=1102.704,-54.355,-49.727,179.871,5.510,149.005
C09976=1102.699,-54.106,-49.740,179.871,5.515,149.006
C09977=1102.693,-53.857,-49.753,179.872,5.520,149.007
C09978=1102.688,-53.607,-49.765,179.871,5.524,149.008
C09979=1102.683,-53.357,-49.777,179.871,5.529,149.010
C09980=1102.678,-53.107,-49.790,179.871,5.534,149.010
C09981=1102.673,-52.857,-49.802,179.871,5.539,149.012
C09982=1102.668,-52.608,-49.815,179.871,5.544,149.013
C09983=1102.663,-52.359,-49.827,179.871,5.548,149.014
C09984=1102.657,-52.109,-49.839,179.870,5.553,149.015
C09985=1102.652,-51.859,-49.852,179.870,5.558,149.016
C09986=1102.648,-51.609,-49.865,179.871,5.563,149.017
C09987=1102.642,-51.360,-49.877,179.870,5.567,149.018
C09988=1102.637,-51.110,-49.889,179.870,5.572,149.019
C09989=1102.632,-50.861,-49.902,179.870,5.577,149.020
C09990=1102.627,-50.611,-49.914,179.870,5.581,149.021
C09991=1102.621,-50.362,-49.926,179.869,5.586,149.022
C09992=1102.617,-50.112,-49.939,179.870,5.591,149.023
C09993=1102.612,-49.862,-49.952,179.869,5.595,149.025
C09994=1102.606,-49.612,-49.964,179.869,5.600,149.026
C09995=1102.601,-49.363,-49.976,179.870,5.605,149.027
C09996=1102.596,-49.114,-49.989,179.869,5.609,149.028
//INST
///DATE 2021/06/25 14:34
///ATTR SC,RW,RJ
////FRAME ROBOT
///GROUP1 RB1
NOP
MOVL C00000 V=800.0 PL=0
MOVL C00001 V=800.0 PL=0
MOVL C00002 V=800.0 PL=0
MOVL C00003 V=800.0 PL=0
MOVL C00004 V=800.0 PL=0
MOVL C00005 V=800.0 PL=0
MOVL C00006 V=800.0 PL=0
MOVL C00007 V=800.0 PL=0
MOVL C00008 V=800.0 PL=0
MOVL C00009 V=800.0 PL=0
MOVL C00010 V=800.0 PL=0
MOVL C00011 V=800.0 PL=0
MOVL C00012 V=800.0 PL=0
MOVL C00013 V=800.0 PL=0
MOVL C00014 V=800.0 PL=0
MOVL C00015 V=800.0 PL=0
MOVL C00016 V=800.0 PL=0
MOVL C00017 V=800.0 PL=0
MOVL C00018 V=800.0 PL=0
MOVL C00019 V=800.0 PL=0
MOVL C00020 V=800.0 PL=0
MOVL C00021 V=800.0 PL=0
MOVL C00022 V=800.0 PL=0
MOVL C00023 V=800.0 PL=0
MOVL C00024 V=800.0 PL=0
MOVL C00025 V=800.0 PL=0
MOVL C00026 V=800.0 PL=0
MOVL C00027 V=800.0 PL=0
MOVL C00028 V=800.0 PL=0
MOVL C00029 V=800.0 PL=0
MOVL C00030 V=800.0 PL=0
MOVL C00031 V=800.0 PL=0
MOVL C00032 V=800.0 PL=0
MOVL C00033 V=800.0 PL=0
MOVL C00034 V=800.0 PL=0
MOVL C00035 V=800.0 PL=0
MOVL C00036 V=800.0 PL=0
MOVL C00037 V=800.0 PL=0
MOVL C00038 V=800.0 PL=0
MOVL C00039 V=800.0 PL=0
MOVL C00040 V=800.0 PL=0
MOVL C00041 V=800.0 PL=0
MOVL C00042 V=800.0 PL=0
MOVL C00043 V=800.0 PL=0
MOVL C00044 V=800.0 PL=0
MOVL C00045 V=800.0 PL=0
MOVL C00046 V=800.0 PL=0
MOVL C00047 V=800.0 PL=0
MOVL C00048 V=800.0 PL=0
MOVL C00049 V=800.0 PL=0
MOVL C00050 V=800.0 PL=0
MOVL C00051 V=800.0 PL=0
MOVL C00052 V=800.0 PL=0
MOVL C00053 V=800.0 PL=0
MOVL C00054 V=800.0 PL=0
MOVL C00055 V=800.0 PL=0
MOVL C00056 V=800.0 PL=0
MOVL C00057 V=800.0 PL=0
MOVL C00058 V=800.0 PL=0
MOVL C00059 V=800.0 PL=0
MOVL C00060 V=800.0 PL=0
MOVL C00061 V=800.0 PL=0
MOVL C00062 V=800.0 PL=0
MOVL C00063 V=800.0 PL=0
MOVL C00064 V=800.0 PL=0
MOVL C00065 V=800.0 PL=0
MOVL C00066 V=800.0 PL=0
MOVL C00067 V=800.0 PL=0
MOVL C00068 V=800.0 PL=0
MOVL C00069 V=800.0 PL=0
MOVL C00070 V=800.0 PL=0
MOVL C00071 V=800.0 PL=0
MOVL C00072 V=800.0 PL=0
MOVL C00073 V=800.0 PL=0
MOVL C00074 V=800.0 PL=0
MOVL C00075 V=800.0 PL=0
MOVL C00076 V=800.0 PL=0
MOVL C00077 V=800.0 PL=0
MOVL C00078 V=800.0 PL=0
MOVL C00079 V=800.0 PL=0
MOVL C00080 V=800.0 PL=0
MOVL C00081 V=800.0 PL=0
MOVL C00082 V=800.0 PL=0
MOVL C00083 V=800.0 PL=0
MOVL C00084 V=800.0 PL=0
MOVL C00085 V=800.0 PL=0
MOVL C00086 V=800.0 PL=0
MOVL C00087 V=800.0 PL=0
MOVL C00088 V=800.0 PL=0
MOVL C00089 V=800.0 PL=0
MOVL C00090 V=800.0 PL=0
MOVL C00091 V=800.0 PL=0
MOVL C00092 V=800.0 PL=0
MOVL C00093 V=800.0 PL=0
MOVL C00094 V=800.0 PL=0
MOVL C00095 V=800.0 PL=0
MOVL C00096 V=800.0 PL=0
MOVL C00097 V=800.0 PL=0
MOVL C00098 V=800.0 PL=0
MOVL C00099 V=800.0 PL=0
MOVL C00100 V=800.0 PL=0
MOVL C00101 V=800.0 PL=0
MOVL C00102 V=800.0 PL=0
MOVL C00103 V=800.0 PL=0
MOVL C00104 V=800.0 PL=0
MOVL C00105 V=800.0 PL=0
MOVL C00106 V=800.0 PL=0
MOVL C00107 V=800.0 PL=0
MOVL C00108 V=800.0 PL=0
MOVL C00109 V=800.0 PL=0
MOVL C00110 V=800.0 PL=0
MOVL C00111 V=800.0 PL=0
MOVL C00112 V=800.0 PL=0
MOVL C00113 V=800.0 PL=0
MOVL C00114 V=800.0 PL=0
MOVL C00115 V=800.0 PL=0
MOVL C00116 V=800.0 PL=0
MOVL C00117 V=800.0 PL=0
MOVL C00118 V=800.0 PL=0
MOVL C00119 V=800.0 PL=0
MOVL C00120 V=800.0 PL=0
MOVL C00121 V=800.0 PL=0
MOVL C00122 V=800.0 PL=0
MOVL C00123 V=800.0 PL=0
MOVL C00124 V=800.0 PL=0
MOVL C00125 V=800.0 PL=0
MOVL C00126 V=800.0 PL=0
MOVL C00127 V=800.0 PL=0
MOVL C00128 V=800.0 PL=0
MOVL C00129 V=800.0 PL=0
MOVL C00130 V=800.0 PL=0
MOVL C00131 V=800.0 PL=0
MOVL C00132 V=800.0 PL=0
MOVL C00133 V=800.0 PL=0
MOVL C00134 V=800.0 PL=0
MOVL C00135 V=800.0 PL=0
MOVL C00136 V=800.0 PL=0
MOVL C00137 V=800.0 PL=0
MOVL C00138 V=800.0 PL=0
MOVL C00139 V=800.0 PL=0
MOVL C00140 V=800.0 PL=0
MOVL C00141 V=800.0 PL=0
MOVL C00142 V=800.0 PL=0
MOVL C00143 V=800.0 PL=0
MOVL C00144 V=800.0 PL=0
MOVL C00145 V=800.0 PL=0
MOVL C00146 V=800.0 PL=0
MOVL C00147 V=800.0 PL=0
MOVL C00148 V=800.0 PL=0
MOVL C00149 V=800.0 PL=0
MOVL C00150 V=800.0 PL=0
MOVL C00151 V=800.0 PL=0
MOVL C00152 V=800.0 PL=0
MOVL C00153 V=800.0 PL=0
MOVL C00154 V=800.0 PL=0
MOVL C00155 V=800.0 PL=0
MOVL C00156 V=800.0 PL=0
MOVL C00157 V=800.0 PL=0
MOVL C00158 V=800.0 PL=0
MOVL C00159 V=800.0 PL=0
MOVL C00160 V=800.0 PL=0
MOVL C00161 V=800.0 PL=0
MOVL C00162 V=800.0 PL=0
MOVL C00163 V=800.0 PL=0
MOVL C00164 V=800.0 PL=0
MOVL C00165 V=800.0 PL=0
MOVL C00166 V=800.0 PL=0
MOVL C00167 V=800.0 PL=0
MOVL C00168 V=800.0 PL=0
MOVL C00169 V=800.0 PL=0
MOVL C00170 V=800.0 PL=0
MOVL C00171 V=800.0 PL=0
MOVL C00172 V=800.0 PL=0
MOVL C00173 V=800.0 PL=0
MOVL C00174 V=800.0 PL=0
MOVL C00175 V=800.0 PL=0
MOVL C00176 V=800.0 PL=0
MOVL C00177 V=800.0 PL=0
MOVL C00178 V=800.0 PL=0
MOVL C00179 V=800.0 PL=0
MOVL C00180 V=800.0 PL=0
MOVL C00181 V=800.0 PL=0
MOVL C00182 V=800.0 PL=0
MOVL C00183 V=800.0 PL=0
MOVL C00184 V=800.0 PL=0
MOVL C00185 V=800.0 PL=0
MOVL C00186 V=800.0 PL=0
MOVL C00187 V=800.0 PL=0
MOVL C00188 V=800.0 PL=0
MOVL C00189 V=800.0 PL=0
MOVL C00190 V=800.0 PL=0
MOVL C00191 V=800.0 PL=0
MOVL C00192 V=800.0 PL=0
MOVL C00193 V=800.0 PL=0
MOVL C00194 V=800.0 PL=0
MOVL C00195 V=800.0 PL=0
MOVL C00196 V=800.0 PL=0
MOVL C00197 V=800.0 PL=0
MOVL C00198 V=800.0 PL=0
MOVL C00199 V=800.0 PL=0
MOVL C00200 V=800.0 PL=0
MOVL C00201 V=800.0 PL=0
MOVL C00202 V=800.0 PL=0
MOVL C00203 V=800.0 PL=0
MOVL C00204 V=800.0 PL=0
MOVL C00205 V=800.0 PL=0
MOVL C00206 V=800.0 PL=0
MOVL C00207 V=800.0 PL=0
MOVL C00208 V=800.0 PL=0
MOVL C00209 V=800.0 PL=0
MOVL C00210 V=800.0 PL=0
MOVL C00211 V=800.0 PL=0
MOVL C00212 V=800.0 PL=0
MOVL C00213 V=800.0 PL=0
MOVL C00214 V=800.0 PL=0
MOVL C00215 V=800.0 PL=0
MOVL C00216 V=800.0 PL=0
MOVL C00217 V=800.0 PL=0
MOVL C00218 V=800.0 PL=0
MOVL C00219 V=800.0 PL=0
MOVL C00220 V=800.0 PL=0
MOVL C00221 V=800.0 PL=0
MOVL C00222 V=800.0 PL=0
MOVL C00223 V=800.0 PL=0
MOVL C00224 V=800.0 PL=0
MOVL C00225 V=800.0 PL=0
MOVL C00226 V=800.0 PL=0
MOVL C00227 V=800.0 PL=0
MOVL C00228 V=800.0 PL=0
MOVL C00229 V=800.0 PL=0
MOVL C00230 V=800.0 PL=0
MOVL C00231 V=800.0 PL=0
MOVL C00232 V=800.0 PL=0
MOVL C00233 V=800.0 PL=0
MOVL C00234 V=800.0 PL=0
MOVL C00235 V=800.0 PL=0
MOVL C00236 V=800.0 PL=0
MOVL C00237 V=800.0 PL=0
MOVL C00238 V=800.0 PL=0
MOVL C00239 V=800.0 PL=0
MOVL C00240 V=800.0 PL=0
MOVL C00241 V=800.0 PL=0
MOVL C00242 V=800.0 PL=0
MOVL C00243 V=800.0 PL=0
MOVL C00244 V=800.0 PL=0
MOVL C00245 V=800.0 PL=0
MOVL C00246 V=800.0 PL=0
MOVL C00247 V=800.0 PL=0
MOVL C00248 V=800.0 PL=0
MOVL C00249 V=800.0 PL=0
MOVL C00250 V=800.0 PL=0
MOVL C00251 V=800.0 PL=0
MOVL C00252 V=800.0 PL=0
MOVL C00253 V=800.0 PL=0
MOVL C00254 V=800.0 PL=0
MOVL C00255 V=800.0 PL=0
MOVL C00256 V=800.0 PL=0
MOVL C00257 V=800.0 PL=0
MOVL C00258 V=800.0 PL=0
MOVL C00259 V=800.0 PL=0
MOVL C00260 V=800.0 PL=0
MOVL C00261 V=800.0 PL=0
MOVL C00262 V=800.0 PL=0
MOVL C00263 V=800.0 PL=0
MOVL C00264 V=800.0 PL=0
MOVL C00265 V=800.0 PL=0
MOVL C00266 V=800.0 PL=0
MOVL C00267 V=800.0 PL=0
MOVL C00268 V=800.0 PL=0
MOVL C00269 V=800.0 PL=0
MOVL C00270 V=800.0 PL=0
MOVL C00271 V=800.0 PL=0
MOVL C00272 V=800.0 PL=0
MOVL C00273 V=800.0 PL=0
MOVL C00274 V=800.0 PL=0
MOVL C00275 V=800.0 PL=0
MOVL C00276 V=800.0 PL=0
MOVL C00277 V=800.0 PL=0
MOVL C00278 V=800.0 PL=0
MOVL C00279 V=800.0 PL=0
MOVL C00280 V=800.0 PL=0
MOVL C00281 V=800.0 PL=0
MOVL C00282 V=800.0 PL=0
MOVL C00283 V=800.0 PL=0
MOVL C00284 V=800.0 PL=0
MOVL C00285 V=800.0 PL=0
MOVL C00286 V=800.0 PL=0
MOVL C00287 V=800.0 PL=0
MOVL C00288 V=800.0 PL=0
MOVL C00289 V=800.0 PL=0
MOVL C00290 V=800.0 PL=0
MOVL C00291 V=800.0 PL=0
MOVL C00292 V=800.0 PL=0
MOVL C00293 V=800.0 PL=0
MOVL C00294 V=800.0 PL=0
MOVL C00295 V=800.0 PL=0
MOVL C00296 V=800.0 PL=0
MOVL C00297 V=800.0 PL=0
MOVL C00298 V=800.0 PL=0
MOVL C00299 V=800.0 PL=0
MOVL C00300 V=800.0 PL=0
MOVL C00301 V=800.0 PL=0
MOVL C00302 V=800.0 PL=0
MOVL C00303 V=800.0 PL=0
MOVL C00304 V=800.0 PL=0
MOVL C00305 V=800.0 PL=0
MOVL C00306 V=800.0 PL=0
MOVL C00307 V=800.0 PL=0
MOVL C00308 V=800.0 PL=0
MOVL C00309 V=800.0 PL=0
MOVL C00310 V=800.0 PL=0
MOVL C00311 V=800.0 PL=0
MOVL C00312 V=800.0 PL=0
MOVL C00313 V=800.0 PL=0
MOVL C00314 V=800.0 PL=0
MOVL C00315 V=800.0 PL=0
MOVL C00316 V=800.0 PL=0
MOVL C00317 V=800.0 PL=0
MOVL C00318 V=800.0 PL=0
MOVL C00319 V=800.0 PL=0
MOVL C00320 V=800.0 PL=0
MOVL C00321 V=800.0 PL=0
MOVL C00322 V=800.0 PL=0
MOVL C00323 V=800.0 PL=0
MOVL C00324 V=800.0 PL=0
MOVL C00325 V=800.0 PL=0
MOVL C00326 V=800.0 PL=0
MOVL C00327 V=800.0 PL=0
MOVL C00328 V=800.0 PL=0
MOVL C00329 V=800.0 PL=0
MOVL C00330 V=800.0 PL=0
MOVL C00331 V=800.0 PL=0
MOVL C00332 V=800.0 PL=0
MOVL C00333 V=800.0 PL=0
MOVL C00334 V=800.0 PL=0
MOVL C00335 V=800.0 PL=0
MOVL C00336 V=800.0 PL=0
MOVL C00337 V=800.0 PL=0
MOVL C00338 V=800.0 PL=0
MOVL C00339 V=800.0 PL=0
MOVL C00340 V=800.0 PL=0
MOVL C00341 V=800.0 PL=0
MOVL C00342 V=800.0 PL=0
MOVL C00343 V=800.0 PL=0
MOVL C00344 V=800.0 PL=0
MOVL C00345 V=800.0 PL=0
MOVL C00346 V=800.0 PL=0
MOVL C00347 V=800.0 PL=0
MOVL C00348 V=800.0 PL=0
MOVL C00349 V=800.0 PL=0
MOVL C00350 V=800.0 PL=0
MOVL C00351 V=800.0 PL=0
MOVL C00352 V=800.0 PL=0
MOVL C00353 V=800.0 PL=0
MOVL C00354 V=800.0 PL=0
MOVL C00355 V=800.0 PL=0
MOVL C00356 V=800.0 PL=0
MOVL C00357 V=800.0 PL=0
MOVL C00358 V=800.0 PL=0
MOVL C00359 V=800.0 PL=0
MOVL C00360 V=800.0 PL=0
MOVL C00361 V=800.0 PL=0
MOVL C00362 V=800.0 PL=0
MOVL C00363 V=800.0 PL=0
MOVL C00364 V=800.0 PL=0
MOVL C00365 V=800.0 PL=0
MOVL C00366 V=800.0 PL=0
MOVL C00367 V=800.0 PL=0
MOVL C00368 V=800.0 PL=0
MOVL C00369 V=800.0 PL=0
MOVL C00370 V=800.0 PL=0
MOVL C00371 V=800.0 PL=0
MOVL C00372 V=800.0 PL=0
MOVL C00373 V=800.0 PL=0
MOVL C00374 V=800.0 PL=0
MOVL C00375 V=800.0 PL=0
MOVL C00376 V=800.0 PL=0
MOVL C00377 V=800.0 PL=0
MOVL C00378 V=800.0 PL=0
MOVL C00379 V=800.0 PL=0
MOVL C00380 V=800.0 PL=0
MOVL C00381 V=800.0 PL=0
MOVL C00382 V=800.0 PL=0
MOVL C00383 V=800.0 PL=0
MOVL C00384 V=800.0 PL=0
MOVL C00385 V=800.0 PL=0
MOVL C00386 V=800.0 PL=0
MOVL C00387 V=800.0 PL=0
MOVL C00388 V=800.0 PL=0
MOVL C00389 V=800.0 PL=0
MOVL C00390 V=800.0 PL=0
MOVL C00391 V=800.0 PL=0
MOVL C00392 V=800.0 PL=0
MOVL C00393 V=800.0 PL=0
MOVL C00394 V=800.0 PL=0
MOVL C00395 V=800.0 PL=0
MOVL C00396 V=800.0 PL=0
MOVL C00397 V=800.0 PL=0
MOVL C00398 V=800.0 PL=0
MOVL C00399 V=800.0 PL=0
MOVL C00400 V=800.0 PL=0
MOVL C00401 V=800.0 PL=0
MOVL C00402 V=800.0 PL=0
MOVL C00403 V=800.0 PL=0
MOVL C00404 V=800.0 PL=0
MOVL C00405 V=800.0 PL=0
MOVL C00406 V=800.0 PL=0
MOVL C00407 V=800.0 PL=0
MOVL C00408 V=800.0 PL=0
MOVL C00409 V=800.0 PL=0
MOVL C00410 V=800.0 PL=0
MOVL C00411 V=800.0 PL=0
MOVL C00412 V=800.0 PL=0
MOVL C00413 V=800.0 PL=0
MOVL C00414 V=800.0 PL=0
MOVL C00415 V=800.0 PL=0
MOVL C00416 V=800.0 PL=0
MOVL C00417 V=800.0 PL=0
MOVL C00418 V=800.0 PL=0
MOVL C00419 V=800.0 PL=0
MOVL C00420 V=800.0 PL=0
MOVL C00421 V=800.0 PL=0
MOVL C00422 V=800.0 PL=0
MOVL C00423 V=800.0 PL=0
MOVL C00424 V=800.0 PL=0
MOVL C00425 V=800.0 PL=0
MOVL C00426 V=800.0 PL=0
MOVL C00427 V=800.0 PL=0
MOVL C00428 V=800.0 PL=0
MOVL C00429 V=800.0 PL=0
MOVL C00430 V=800.0 PL=0
MOVL C00431 V=800.0 PL=0
MOVL C00432 V=800.0 PL=0
MOVL C00433 V=800.0 PL=0
MOVL C00434 V=800.0 PL=0
MOVL C00435 V=800.0 PL=0
MOVL C00436 V=800.0 PL=0
MOVL C00437 V=800.0 PL=0
MOVL C00438 V=800.0 PL=0
MOVL C00439 V=800.0 PL=0
MOVL C00440 V=800.0 PL=0
MOVL C00441 V=800.0 PL=0
MOVL C00442 V=800.0 PL=0
MOVL C00443 V=800.0 PL=0
MOVL C00444 V=800.0 PL=0
MOVL C00445 V=800.0 PL=0
MOVL C00446 V=800.0 PL=0
MOVL C00447 V=800.0 PL=0
MOVL C00448 V=800.0 PL=0
MOVL C00449 V=800.0 PL=0
MOVL C00450 V=800.0 PL=0
MOVL C00451 V=800.0 PL=0
MOVL C00452 V=800.0 PL=0
MOVL C00453 V=800.0 PL=0
MOVL C00454 V=800.0 PL=0
MOVL C00455 V=800.0 PL=0
MOVL C00456 V=800.0 PL=0
MOVL C00457 V=800.0 PL=0
MOVL C00458 V=800.0 PL=0
MOVL C00459 V=800.0 PL=0
MOVL C00460 V=800.0 PL=0
MOVL C00461 V=800.0 PL=0
MOVL C00462 V=800.0 PL=0
MOVL C00463 V=800.0 PL=0
MOVL C00464 V=800.0 PL=0
MOVL C00465 V=800.0 PL=0
MOVL C00466 V=800.0 PL=0
MOVL C00467 V=800.0 PL=0
MOVL C00468 V=800.0 PL=0
MOVL C00469 V=800.0 PL=0
MOVL C00470 V=800.0 PL=0
MOVL C00471 V=800.0 PL=0
MOVL C00472 V=800.0 PL=0
MOVL C00473 V=800.0 PL=0
MOVL C00474 V=800.0 PL=0
MOVL C00475 V=800.0 PL=0
MOVL C00476 V=800.0 PL=0
MOVL C00477 V=800.0 PL=0
MOVL C00478 V=800.0 PL=0
MOVL C00479 V=800.0 PL=0
MOVL C00480 V=800.0 PL=0
MOVL C00481 V=800.0 PL=0
MOVL C00482 V=800.0 PL=0
MOVL C00483 V=800.0 PL=0
MOVL C00484 V=800.0 PL=0
MOVL C00485 V=800.0 PL=0
MOVL C00486 V=800.0 PL=0
MOVL C00487 V=800.0 PL=0
MOVL C00488 V=800.0 PL=0
MOVL C00489 V=800.0 PL=0
MOVL C00490 V=800.0 PL=0
MOVL C00491 V=800.0 PL=0
MOVL C00492 V=800.0 PL=0
MOVL C00493 V=800.0 PL=0
MOVL C00494 V=800.0 PL=0
MOVL C00495 V=800.0 PL=0
MOVL C00496 V=800.0 PL=0
MOVL C00497 V=800.0 PL=0
MOVL C00498 V=800.0 PL=0
MOVL C00499 V=800.0 PL=0
MOVL C00500 V=800.0 PL=0
MOVL C00501 V=800.0 PL=0
MOVL C00502 V=800.0 PL=0
MOVL C00503 V=800.0 PL=0
MOVL C00504 V=800.0 PL=0
MOVL C00505 V=800.0 PL=0
MOVL C00506 V=800.0 PL=0
MOVL C00507 V=800.0 PL=0
MOVL C00508 V=800.0 PL=0
MOVL C00509 V=800.0 PL=0
MOVL C00510 V=800.0 PL=0
MOVL C00511 V=800.0 PL=0
MOVL C00512 V=800.0 PL=0
MOVL C00513 V=800.0 PL=0
MOVL C00514 V=800.0 PL=0
MOVL C00515 V=800.0 PL=0
MOVL C00516 V=800.0 PL=0
MOVL C00517 V=800.0 PL=0
MOVL C00518 V=800.0 PL=0
MOVL C00519 V=800.0 PL=0
MOVL C00520 V=800.0 PL=0
MOVL C00521 V=800.0 PL=0
MOVL C00522 V=800.0 PL=0
MOVL C00523 V=800.0 PL=0
MOVL C00524 V=800.0 PL=0
MOVL C00525 V=800.0 PL=0
MOVL C00526 V=800.0 PL=0
MOVL C00527 V=800.0 PL=0
MOVL C00528 V=800.0 PL=0
MOVL C00529 V=800.0 PL=0
MOVL C00530 V=800.0 PL=0
MOVL C00531 V=800.0 PL=0
MOVL C00532 V=800.0 PL=0
MOVL C00533 V=800.0 PL=0
MOVL C00534 V=800.0 PL=0
MOVL C00535 V=800.0 PL=0
MOVL C00536 V=800.0 PL=0
MOVL C00537 V=800.0 PL=0
MOVL C00538 V=800.0 PL=0
MOVL C00539 V=800.0 PL=0
MOVL C00540 V=800.0 PL=0
MOVL C00541 V=800.0 PL=0
MOVL C00542 V=800.0 PL=0
MOVL C00543 V=800.0 PL=0
MOVL C00544 V=800.0 PL=0
MOVL C00545 V=800.0 PL=0
MOVL C00546 V=800.0 PL=0
MOVL C00547 V=800.0 PL=0
MOVL C00548 V=800.0 PL=0
MOVL C00549 V=800.0 PL=0
MOVL C00550 V=800.0 PL=0
MOVL C00551 V=800.0 PL=0
MOVL C00552 V=800.0 PL=0
MOVL C00553 V=800.0 PL=0
MOVL C00554 V=800.0 PL=0
MOVL C00555 V=800.0 PL=0
MOVL C00556 V=800.0 PL=0
MOVL C00557 V=800.0 PL=0
MOVL C00558 V=800.0 PL=0
MOVL C00559 V=800.0 PL=0
MOVL C00560 V=800.0 PL=0
MOVL C00561 V=800.0 PL=0
MOVL C00562 V=800.0 PL=0
MOVL C00563 V=800.0 PL=0
MOVL C00564 V=800.0 PL=0
MOVL C00565 V=800.0 PL=0
MOVL C00566 V=800.0 PL=0
MOVL C00567 V=800.0 PL=0
MOVL C00568 V=800.0 PL=0
MOVL C00569 V=800.0 PL=0
MOVL C00570 V=800.0 PL=0
MOVL C00571 V=800.0 PL=0
MOVL C00572 V=800.0 PL=0
MOVL C00573 V=800.0 PL=0
MOVL C00574 V=800.0 PL=0
MOVL C00575 V=800.0 PL=0
MOVL C00576 V=800.0 PL=0
MOVL C00577 V=800.0 PL=0
MOVL C00578 V=800.0 PL=0
MOVL C00579 V=800.0 PL=0
MOVL C00580 V=800.0 PL=0
MOVL C00581 V=800.0 PL=0
MOVL C00582 V=800.0 PL=0
MOVL C00583 V=800.0 PL=0
MOVL C00584 V=800.0 PL=0
MOVL C00585 V=800.0 PL=0
MOVL C00586 V=800.0 PL=0
MOVL C00587 V=800.0 PL=0
MOVL C00588 V=800.0 PL=0
MOVL C00589 V=800.0 PL=0
MOVL C00590 V=800.0 PL=0
MOVL C00591 V=800.0 PL=0
MOVL C00592 V=800.0 PL=0
MOVL C00593 V=800.0 PL=0
MOVL C00594 V=800.0 PL=0
MOVL C00595 V=800.0 PL=0
MOVL C00596 V=800.0 PL=0
MOVL C00597 V=800.0 PL=0
MOVL C00598 V=800.0 PL=0
MOVL C00599 V=800.0 PL=0
MOVL C00600 V=800.0 PL=0
MOVL C00601 V=800.0 PL=0
MOVL C00602 V=800.0 PL=0
MOVL C00603 V=800.0 PL=0
MOVL C00604 V=800.0 PL=0
MOVL C00605 V=800.0 PL=0
MOVL C00606 V=800.0 PL=0
MOVL C00607 V=800.0 PL=0
MOVL C00608 V=800.0 PL=0
MOVL C00609 V=800.0 PL=0
MOVL C00610 V=800.0 PL=0
MOVL C00611 V=800.0 PL=0
MOVL C00612 V=800.0 PL=0
MOVL C00613 V=800.0 PL=0
MOVL C00614 V=800.0 PL=0
MOVL C00615 V=800.0 PL=0
MOVL C00616 V=800.0 PL=0
MOVL C00617 V=800.0 PL=0
MOVL C00618 V=800.0 PL=0
MOVL C00619 V=800.0 PL=0
MOVL C00620 V=800.0 PL=0
MOVL C00621 V=800.0 PL=0
MOVL C00622 V=800.0 PL=0
MOVL C00623 V=800.0 PL=0
MOVL C00624 V=800.0 PL=0
MOVL C00625 V=800.0 PL=0
MOVL C00626 V=800.0 PL=0
MOVL C00627 V=800.0 PL=0
MOVL C00628 V=800.0 PL=0
MOVL C00629 V=800.0 PL=0
MOVL C00630 V=800.0 PL=0
MOVL C00631 V=800.0 PL=0
MOVL C00632 V=800.0 PL=0
MOVL C00633 V=800.0 PL=0
MOVL C00634 V=800.0 PL=0
MOVL C00635 V=800.0 PL=0
MOVL C00636 V=800.0 PL=0
MOVL C00637 V=800.0 PL=0
MOVL C00638 V=800.0 PL=0
MOVL C00639 V=800.0 PL=0
MOVL C00640 V=800.0 PL=0
MOVL C00641 V=800.0 PL=0
MOVL C00642 V=800.0 PL=0
MOVL C00643 V=800.0 PL=0
MOVL C00644 V=800.0 PL=0
MOVL C00645 V=800.0 PL=0
MOVL C00646 V=800.0 PL=0
MOVL C00647 V=800.0 PL=0
MOVL C00648 V=800.0 PL=0
MOVL C00649 V=800.0 PL=0
MOVL C00650 V=800.0 PL=0
MOVL C00651 V=800.0 PL=0
MOVL C00652 V=800.0 PL=0
MOVL C00653 V=800.0 PL=0
MOVL C00654 V=800.0 PL=0
MOVL C00655 V=800.0 PL=0
MOVL C00656 V=800.0 PL=0
MOVL C00657 V=800.0 PL=0
MOVL C00658 V=800.0 PL=0
MOVL C00659 V=800.0 PL=0
MOVL C00660 V=800.0 PL=0
MOVL C00661 V=800.0 PL=0
MOVL C00662 V=800.0 PL=0
MOVL C00663 V=800.0 PL=0
MOVL C00664 V=800.0 PL=0
MOVL C00665 V=800.0 PL=0
MOVL C00666 V=800.0 PL=0
MOVL C00667 V=800.0 PL=0
MOVL C00668 V=800.0 PL=0
MOVL C00669 V=800.0 PL=0
MOVL C00670 V=800.0 PL=0
MOVL C00671 V=800.0 PL=0
MOVL C00672 V=800.0 PL=0
MOVL C00673 V=800.0 PL=0
MOVL C00674 V=800.0 PL=0
MOVL C00675 V=800.0 PL=0
MOVL C00676 V=800.0 PL=0
MOVL C00677 V=800.0 PL=0
MOVL C00678 V=800.0 PL=0
MOVL C00679 V=800.0 PL=0
MOVL C00680 V=800.0 PL=0
MOVL C00681 V=800.0 PL=0
MOVL C00682 V=800.0 PL=0
MOVL C00683 V=800.0 PL=0
MOVL C00684 V=800.0 PL=0
MOVL C00685 V=800.0 PL=0
MOVL C00686 V=800.0 PL=0
MOVL C00687 V=800.0 PL=0
MOVL C00688 V=800.0 PL=0
MOVL C00689 V=800.0 PL=0
MOVL C00690 V=800.0 PL=0
MOVL C00691 V=800.0 PL=0
MOVL C00692 V=800.0 PL=0
MOVL C00693 V=800.0 PL=0
MOVL C00694 V=800.0 PL=0
MOVL C00695 V=800.0 PL=0
MOVL C00696 V=800.0 PL=0
MOVL C00697 V=800.0 PL=0
MOVL C00698 V=800.0 PL=0
MOVL C00699 V=800.0 PL=0
MOVL C00700 V=800.0 PL=0
MOVL C00701 V=800.0 PL=0
MOVL C00702 V=800.0 PL=0
MOVL C00703 V=800.0 PL=0
MOVL C00704 V=800.0 PL=0
MOVL C00705 V=800.0 PL=0
MOVL C00706 V=800.0 PL=0
MOVL C00707 V=800.0 PL=0
MOVL C00708 V=800.0 PL=0
MOVL C00709 V=800.0 PL=0
MOVL C00710 V=800.0 PL=0
MOVL C00711 V=800.0 PL=0
MOVL C00712 V=800.0 PL=0
MOVL C00713 V=800.0 PL=0
MOVL C00714 V=800.0 PL=0
MOVL C00715 V=800.0 PL=0
MOVL C00716 V=800.0 PL=0
MOVL C00717 V=800.0 PL=0
MOVL C00718 V=800.0 PL=0
MOVL C00719 V=800.0 PL=0
MOVL C00720 V=800.0 PL=0
MOVL C00721 V=800.0 PL=0
MOVL C00722 V=800.0 PL=0
MOVL C00723 V=800.0 PL=0
MOVL C00724 V=800.0 PL=0
MOVL C00725 V=800.0 PL=0
MOVL C00726 V=800.0 PL=0
MOVL C00727 V=800.0 PL=0
MOVL C00728 V=800.0 PL=0
MOVL C00729 V=800.0 PL=0
MOVL C00730 V=800.0 PL=0
MOVL C00731 V=800.0 PL=0
MOVL C00732 V=800.0 PL=0
MOVL C00733 V=800.0 PL=0
MOVL C00734 V=800.0 PL=0
MOVL C00735 V=800.0 PL=0
MOVL C00736 V=800.0 PL=0
MOVL C00737 V=800.0 PL=0
MOVL C00738 V=800.0 PL=0
MOVL C00739 V=800.0 PL=0
MOVL C00740 V=800.0 PL=0
MOVL C00741 V=800.0 PL=0
MOVL C00742 V=800.0 PL=0
MOVL C00743 V=800.0 PL=0
MOVL C00744 V=800.0 PL=0
MOVL C00745 V=800.0 PL=0
MOVL C00746 V=800.0 PL=0
MOVL C00747 V=800.0 PL=0
MOVL C00748 V=800.0 PL=0
MOVL C00749 V=800.0 PL=0
MOVL C00750 V=800.0 PL=0
MOVL C00751 V=800.0 PL=0
MOVL C00752 V=800.0 PL=0
MOVL C00753 V=800.0 PL=0
MOVL C00754 V=800.0 PL=0
MOVL C00755 V=800.0 PL=0
MOVL C00756 V=800.0 PL=0
MOVL C00757 V=800.0 PL=0
MOVL C00758 V=800.0 PL=0
MOVL C00759 V=800.0 PL=0
MOVL C00760 V=800.0 PL=0
MOVL C00761 V=800.0 PL=0
MOVL C00762 V=800.0 PL=0
MOVL C00763 V=800.0 PL=0
MOVL C00764 V=800.0 PL=0
MOVL C00765 V=800.0 PL=0
MOVL C00766 V=800.0 PL=0
MOVL C00767 V=800.0 PL=0
MOVL C00768 V=800.0 PL=0
MOVL C00769 V=800.0 PL=0
MOVL C00770 V=800.0 PL=0
MOVL C00771 V=800.0 PL=0
MOVL C00772 V=800.0 PL=0
MOVL C00773 V=800.0 PL=0
MOVL C00774 V=800.0 PL=0
MOVL C00775 V=800.0 PL=0
MOVL C00776 V=800.0 PL=0
MOVL C00777 V=800.0 PL=0
MOVL C00778 V=800.0 PL=0
MOVL C00779 V=800.0 PL=0
MOVL C00780 V=800.0 PL=0
MOVL C00781 V=800.0 PL=0
MOVL C00782 V=800.0 PL=0
MOVL C00783 V=800.0 PL=0
MOVL C00784 V=800.0 PL=0
MOVL C00785 V=800.0 PL=0
MOVL C00786 V=800.0 PL=0
MOVL C00787 V=800.0 PL=0
MOVL C00788 V=800.0 PL=0
MOVL C00789 V=800.0 PL=0
MOVL C00790 V=800.0 PL=0
MOVL C00791 V=800.0 PL=0
MOVL C00792 V=800.0 PL=0
MOVL C00793 V=800.0 PL=0
MOVL C00794 V=800.0 PL=0
MOVL C00795 V=800.0 PL=0
MOVL C00796 V=800.0 PL=0
MOVL C00797 V=800.0 PL=0
MOVL C00798 V=800.0 PL=0
MOVL C00799 V=800.0 PL=0
MOVL C00800 V=800.0 PL=0
MOVL C00801 V=800.0 PL=0
MOVL C00802 V=800.0 PL=0
MOVL C00803 V=800.0 PL=0
MOVL C00804 V=800.0 PL=0
MOVL C00805 V=800.0 PL=0
MOVL C00806 V=800.0 PL=0
MOVL C00807 V=800.0 PL=0
MOVL C00808 V=800.0 PL=0
MOVL C00809 V=800.0 PL=0
MOVL C00810 V=800.0 PL=0
MOVL C00811 V=800.0 PL=0
MOVL C00812 V=800.0 PL=0
MOVL C00813 V=800.0 PL=0
MOVL C00814 V=800.0 PL=0
MOVL C00815 V=800.0 PL=0
MOVL C00816 V=800.0 PL=0
MOVL C00817 V=800.0 PL=0
MOVL C00818 V=800.0 PL=0
MOVL C00819 V=800.0 PL=0
MOVL C00820 V=800.0 PL=0
MOVL C00821 V=800.0 PL=0
MOVL C00822 V=800.0 PL=0
MOVL C00823 V=800.0 PL=0
MOVL C00824 V=800.0 PL=0
MOVL C00825 V=800.0 PL=0
MOVL C00826 V=800.0 PL=0
MOVL C00827 V=800.0 PL=0
MOVL C00828 V=800.0 PL=0
MOVL C00829 V=800.0 PL=0
MOVL C00830 V=800.0 PL=0
MOVL C00831 V=800.0 PL=0
MOVL C00832 V=800.0 PL=0
MOVL C00833 V=800.0 PL=0
MOVL C00834 V=800.0 PL=0
MOVL C00835 V=800.0 PL=0
MOVL C00836 V=800.0 PL=0
MOVL C00837 V=800.0 PL=0
MOVL C00838 V=800.0 PL=0
MOVL C00839 V=800.0 PL=0
MOVL C00840 V=800.0 PL=0
MOVL C00841 V=800.0 PL=0
MOVL C00842 V=800.0 PL=0
MOVL C00843 V=800.0 PL=0
MOVL C00844 V=800.0 PL=0
MOVL C00845 V=800.0 PL=0
MOVL C00846 V=800.0 PL=0
MOVL C00847 V=800.0 PL=0
MOVL C00848 V=800.0 PL=0
MOVL C00849 V=800.0 PL=0
MOVL C00850 V=800.0 PL=0
MOVL C00851 V=800.0 PL=0
MOVL C00852 V=800.0 PL=0
MOVL C00853 V=800.0 PL=0
MOVL C00854 V=800.0 PL=0
MOVL C00855 V=800.0 PL=0
MOVL C00856 V=800.0 PL=0
MOVL C00857 V=800.0 PL=0
MOVL C00858 V=800.0 PL=0
MOVL C00859 V=800.0 PL=0
MOVL C00860 V=800.0 PL=0
MOVL C00861 V=800.0 PL=0
MOVL C00862 V=800.0 PL=0
MOVL C00863 V=800.0 PL=0
MOVL C00864 V=800.0 PL=0
MOVL C00865 V=800.0 PL=0
MOVL C00866 V=800.0 PL=0
MOVL C00867 V=800.0 PL=0
MOVL C00868 V=800.0 PL=0
MOVL C00869 V=800.0 PL=0
MOVL C00870 V=800.0 PL=0
MOVL C00871 V=800.0 PL=0
MOVL C00872 V=800.0 PL=0
MOVL C00873 V=800.0 PL=0
MOVL C00874 V=800.0 PL=0
MOVL C00875 V=800.0 PL=0
MOVL C00876 V=800.0 PL=0
MOVL C00877 V=800.0 PL=0
MOVL C00878 V=800.0 PL=0
MOVL C00879 V=800.0 PL=0
MOVL C00880 V=800.0 PL=0
MOVL C00881 V=800.0 PL=0
MOVL C00882 V=800.0 PL=0
MOVL C00883 V=800.0 PL=0
MOVL C00884 V=800.0 PL=0
MOVL C00885 V=800.0 PL=0
MOVL C00886 V=800.0 PL=0
MOVL C00887 V=800.0 PL=0
MOVL C00888 V=800.0 PL=0
MOVL C00889 V=800.0 PL=0
MOVL C00890 V=800.0 PL=0
MOVL C00891 V=800.0 PL=0
MOVL C00892 V=800.0 PL=0
MOVL C00893 V=800.0 PL=0
MOVL C00894 V=800.0 PL=0
MOVL C00895 V=800.0 PL=0
MOVL C00896 V=800.0 PL=0
MOVL C00897 V=800.0 PL=0
MOVL C00898 V=800.0 PL=0
MOVL C00899 V=800.0 PL=0
MOVL C00900 V=800.0 PL=0
MOVL C00901 V=800.0 PL=0
MOVL C00902 V=800.0 PL=0
MOVL C00903 V=800.0 PL=0
MOVL C00904 V=800.0 PL=0
MOVL C00905 V=800.0 PL=0
MOVL C00906 V=800.0 PL=0
MOVL C00907 V=800.0 PL=0
MOVL C00908 V=800.0 PL=0
MOVL C00909 V=800.0 PL=0
MOVL C00910 V=800.0 PL=0
MOVL C00911 V=800.0 PL=0
MOVL C00912 V=800.0 PL=0
MOVL C00913 V=800.0 PL=0
MOVL C00914 V=800.0 PL=0
MOVL C00915 V=800.0 PL=0
MOVL C00916 V=800.0 PL=0
MOVL C00917 V=800.0 PL=0
MOVL C00918 V=800.0 PL=0
MOVL C00919 V=800.0 PL=0
MOVL C00920 V=800.0 PL=0
MOVL C00921 V=800.0 PL=0
MOVL C00922 V=800.0 PL=0
MOVL C00923 V=800.0 PL=0
MOVL C00924 V=800.0 PL=0
MOVL C00925 V=800.0 PL=0
MOVL C00926 V=800.0 PL=0
MOVL C00927 V=800.0 PL=0
MOVL C00928 V=800.0 PL=0
MOVL C00929 V=800.0 PL=0
MOVL C00930 V=800.0 PL=0
MOVL C00931 V=800.0 PL=0
MOVL C00932 V=800.0 PL=0
MOVL C00933 V=800.0 PL=0
MOVL C00934 V=800.0 PL=0
MOVL C00935 V=800.0 PL=0
MOVL C00936 V=800.0 PL=0
MOVL C00937 V=800.0 PL=0
MOVL C00938 V=800.0 PL=0
MOVL C00939 V=800.0 PL=0
MOVL C00940 V=800.0 PL=0
MOVL C00941 V=800.0 PL=0
MOVL C00942 V=800.0 PL=0
MOVL C00943 V=800.0 PL=0
MOVL C00944 V=800.0 PL=0
MOVL C00945 V=800.0 PL=0
MOVL C00946 V=800.0 PL=0
MOVL C00947 V=800.0 PL=0
MOVL C00948 V=800.0 PL=0
MOVL C00949 V=800.0 PL=0
MOVL C00950 V=800.0 PL=0
MOVL C00951 V=800.0 PL=0
MOVL C00952 V=800.0 PL=0
MOVL C00953 V=800.0 PL=0
MOVL C00954 V=800.0 PL=0
MOVL C00955 V=800.0 PL=0
MOVL C00956 V=800.0 PL=0
MOVL C00957 V=800.0 PL=0
MOVL C00958 V=800.0 PL=0
MOVL C00959 V=800.0 PL=0
MOVL C00960 V=800.0 PL=0
MOVL C00961 V=800.0 PL=0
MOVL C00962 V=800.0 PL=0
MOVL C00963 V=800.0 PL=0
MOVL C00964 V=800.0 PL=0
MOVL C00965 V=800.0 PL=0
MOVL C00966 V=800.0 PL=0
MOVL C00967 V=800.0 PL=0
MOVL C00968 V=800.0 PL=0
MOVL C00969 V=800.0 PL=0
MOVL C00970 V=800.0 PL=0
MOVL C00971 V=800.0 PL=0
MOVL C00972 V=800.0 PL=0
MOVL C00973 V=800.0 PL=0
MOVL C00974 V=800.0 PL=0
MOVL C00975 V=800.0 PL=0
MOVL C00976 V=800.0 PL=0
MOVL C00977 V=800.0 PL=0
MOVL C00978 V=800.0 PL=0
MOVL C00979 V=800.0 PL=0
MOVL C00980 V=800.0 PL=0
MOVL C00981 V=800.0 PL=0
MOVL C00982 V=800.0 PL=0
MOVL C00983 V=800.0 PL=0
MOVL C00984 V=800.0 PL=0
MOVL C00985 V=800.0 PL=0
MOVL C00986 V=800.0 PL=0
MOVL C00987 V=800.0 PL=0
MOVL C00988 V=800.0 PL=0
MOVL C00989 V=800.0 PL=0
MOVL C00990 V=800.0 PL=0
MOVL C00991 V=800.0 PL=0
MOVL C00992 V=800.0 PL=0
MOVL C00993 V=800.0 PL=0
MOVL C00994 V=800.0 PL=0
MOVL C00995 V=800.0 PL=0
MOVL C00996 V=800.0 PL=0
MOVL C00997 V=800.0 PL=0
MOVL C00998 V=800.0 PL=0
MOVL C00999 V=800.0 PL=0
MOVL C01000 V=800.0 PL=0
MOVL C01001 V=800.0 PL=0
MOVL C01002 V=800.0 PL=0
MOVL C01003 V=800.0 PL=0
MOVL C01004 V=800.0 PL=0
MOVL C01005 V=800.0 PL=0
MOVL C01006 V=800.0 PL=0
MOVL C01007 V=800.0 PL=0
MOVL C01008 V=800.0 PL=0
MOVL C01009 V=800.0 PL=0
MOVL C01010 V=800.0 PL=0
MOVL C01011 V=800.0 PL=0
MOVL C01012 V=800.0 PL=0
MOVL C01013 V=800.0 PL=0
MOVL C01014 V=800.0 PL=0
MOVL C01015 V=800.0 PL=0
MOVL C01016 V=800.0 PL=0
MOVL C01017 V=800.0 PL=0
MOVL C01018 V=800.0 PL=0
MOVL C01019 V=800.0 PL=0
MOVL C01020 V=800.0 PL=0
MOVL C01021 V=800.0 PL=0
MOVL C01022 V=800.0 PL=0
MOVL C01023 V=800.0 PL=0
MOVL C01024 V=800.0 PL=0
MOVL C01025 V=800.0 PL=0
MOVL C01026 V=800.0 PL=0
MOVL C01027 V=800.0 PL=0
MOVL C01028 V=800.0 PL=0
MOVL C01029 V=800.0 PL=0
MOVL C01030 V=800.0 PL=0
MOVL C01031 V=800.0 PL=0
MOVL C01032 V=800.0 PL=0
MOVL C01033 V=800.0 PL=0
MOVL C01034 V=800.0 PL=0
MOVL C01035 V=800.0 PL=0
MOVL C01036 V=800.0 PL=0
MOVL C01037 V=800.0 PL=0
MOVL C01038 V=800.0 PL=0
MOVL C01039 V=800.0 PL=0
MOVL C01040 V=800.0 PL=0
MOVL C01041 V=800.0 PL=0
MOVL C01042 V=800.0 PL=0
MOVL C01043 V=800.0 PL=0
MOVL C01044 V=800.0 PL=0
MOVL C01045 V=800.0 PL=0
MOVL C01046 V=800.0 PL=0
MOVL C01047 V=800.0 PL=0
MOVL C01048 V=800.0 PL=0
MOVL C01049 V=800.0 PL=0
MOVL C01050 V=800.0 PL=0
MOVL C01051 V=800.0 PL=0
MOVL C01052 V=800.0 PL=0
MOVL C01053 V=800.0 PL=0
MOVL C01054 V=800.0 PL=0
MOVL C01055 V=800.0 PL=0
MOVL C01056 V=800.0 PL=0
MOVL C01057 V=800.0 PL=0
MOVL C01058 V=800.0 PL=0
MOVL C01059 V=800.0 PL=0
MOVL C01060 V=800.0 PL=0
MOVL C01061 V=800.0 PL=0
MOVL C01062 V=800.0 PL=0
MOVL C01063 V=800.0 PL=0
MOVL C01064 V=800.0 PL=0
MOVL C01065 V=800.0 PL=0
MOVL C01066 V=800.0 PL=0
MOVL C01067 V=800.0 PL=0
MOVL C01068 V=800.0 PL=0
MOVL C01069 V=800.0 PL=0
MOVL C01070 V=800.0 PL=0
MOVL C01071 V=800.0 PL=0
MOVL C01072 V=800.0 PL=0
MOVL C01073 V=800.0 PL=0
MOVL C01074 V=800.0 PL=0
MOVL C01075 V=800.0 PL=0
MOVL C01076 V=800.0 PL=0
MOVL C01077 V=800.0 PL=0
MOVL C01078 V=800.0 PL=0
MOVL C01079 V=800.0 PL=0
MOVL C01080 V=800.0 PL=0
MOVL C01081 V=800.0 PL=0
MOVL C01082 V=800.0 PL=0
MOVL C01083 V=800.0 PL=0
MOVL C01084 V=800.0 PL=0
MOVL C01085 V=800.0 PL=0
MOVL C01086 V=800.0 PL=0
MOVL C01087 V=800.0 PL=0
MOVL C01088 V=800.0 PL=0
MOVL C01089 V=800.0 PL=0
MOVL C01090 V=800.0 PL=0
MOVL C01091 V=800.0 PL=0
MOVL C01092 V=800.0 PL=0
MOVL C01093 V=800.0 PL=0
MOVL C01094 V=800.0 PL=0
MOVL C01095 V=800.0 PL=0
MOVL C01096 V=800.0 PL=0
MOVL C01097 V=800.0 PL=0
MOVL C01098 V=800.0 PL=0
MOVL C01099 V=800.0 PL=0
MOVL C01100 V=800.0 PL=0
MOVL C01101 V=800.0 PL=0
MOVL C01102 V=800.0 PL=0
MOVL C01103 V=800.0 PL=0
MOVL C01104 V=800.0 PL=0
MOVL C01105 V=800.0 PL=0
MOVL C01106 V=800.0 PL=0
MOVL C01107 V=800.0 PL=0
MOVL C01108 V=800.0 PL=0
MOVL C01109 V=800.0 PL=0
MOVL C01110 V=800.0 PL=0
MOVL C01111 V=800.0 PL=0
MOVL C01112 V=800.0 PL=0
MOVL C01113 V=800.0 PL=0
MOVL C01114 V=800.0 PL=0
MOVL C01115 V=800.0 PL=0
MOVL C01116 V=800.0 PL=0
MOVL C01117 V=800.0 PL=0
MOVL C01118 V=800.0 PL=0
MOVL C01119 V=800.0 PL=0
MOVL C01120 V=800.0 PL=0
MOVL C01121 V=800.0 PL=0
MOVL C01122 V=800.0 PL=0
MOVL C01123 V=800.0 PL=0
MOVL C01124 V=800.0 PL=0
MOVL C01125 V=800.0 PL=0
MOVL C01126 V=800.0 PL=0
MOVL C01127 V=800.0 PL=0
MOVL C01128 V=800.0 PL=0
MOVL C01129 V=800.0 PL=0
MOVL C01130 V=800.0 PL=0
MOVL C01131 V=800.0 PL=0
MOVL C01132 V=800.0 PL=0
MOVL C01133 V=800.0 PL=0
MOVL C01134 V=800.0 PL=0
MOVL C01135 V=800.0 PL=0
MOVL C01136 V=800.0 PL=0
MOVL C01137 V=800.0 PL=0
MOVL C01138 V=800.0 PL=0
MOVL C01139 V=800.0 PL=0
MOVL C01140 V=800.0 PL=0
MOVL C01141 V=800.0 PL=0
MOVL C01142 V=800.0 PL=0
MOVL C01143 V=800.0 PL=0
MOVL C01144 V=800.0 PL=0
MOVL C01145 V=800.0 PL=0
MOVL C01146 V=800.0 PL=0
MOVL C01147 V=800.0 PL=0
MOVL C01148 V=800.0 PL=0
MOVL C01149 V=800.0 PL=0
MOVL C01150 V=800.0 PL=0
MOVL C01151 V=800.0 PL=0
MOVL C01152 V=800.0 PL=0
MOVL C01153 V=800.0 PL=0
MOVL C01154 V=800.0 PL=0
MOVL C01155 V=800.0 PL=0
MOVL C01156 V=800.0 PL=0
MOVL C01157 V=800.0 PL=0
MOVL C01158 V=800.0 PL=0
MOVL C01159 V=800.0 PL=0
MOVL C01160 V=800.0 PL=0
MOVL C01161 V=800.0 PL=0
MOVL C01162 V=800.0 PL=0
MOVL C01163 V=800.0 PL=0
MOVL C01164 V=800.0 PL=0
MOVL C01165 V=800.0 PL=0
MOVL C01166 V=800.0 PL=0
MOVL C01167 V=800.0 PL=0
MOVL C01168 V=800.0 PL=0
MOVL C01169 V=800.0 PL=0
MOVL C01170 V=800.0 PL=0
MOVL C01171 V=800.0 PL=0
MOVL C01172 V=800.0 PL=0
MOVL C01173 V=800.0 PL=0
MOVL C01174 V=800.0 PL=0
MOVL C01175 V=800.0 PL=0
MOVL C01176 V=800.0 PL=0
MOVL C01177 V=800.0 PL=0
MOVL C01178 V=800.0 PL=0
MOVL C01179 V=800.0 PL=0
MOVL C01180 V=800.0 PL=0
MOVL C01181 V=800.0 PL=0
MOVL C01182 V=800.0 PL=0
MOVL C01183 V=800.0 PL=0
MOVL C01184 V=800.0 PL=0
MOVL C01185 V=800.0 PL=0
MOVL C01186 V=800.0 PL=0
MOVL C01187 V=800.0 PL=0
MOVL C01188 V=800.0 PL=0
MOVL C01189 V=800.0 PL=0
MOVL C01190 V=800.0 PL=0
MOVL C01191 V=800.0 PL=0
MOVL C01192 V=800.0 PL=0
MOVL C01193 V=800.0 PL=0
MOVL C01194 V=800.0 PL=0
MOVL C01195 V=800.0 PL=0
MOVL C01196 V=800.0 PL=0
MOVL C01197 V=800.0 PL=0
MOVL C01198 V=800.0 PL=0
MOVL C01199 V=800.0 PL=0
MOVL C01200 V=800.0 PL=0
MOVL C01201 V=800.0 PL=0
MOVL C01202 V=800.0 PL=0
MOVL C01203 V=800.0 PL=0
MOVL C01204 V=800.0 PL=0
MOVL C01205 V=800.0 PL=0
MOVL C01206 V=800.0 PL=0
MOVL C01207 V=800.0 PL=0
MOVL C01208 V=800.0 PL=0
MOVL C01209 V=800.0 PL=0
MOVL C01210 V=800.0 PL=0
MOVL C01211 V=800.0 PL=0
MOVL C01212 V=800.0 PL=0
MOVL C01213 V=800.0 PL=0
MOVL C01214 V=800.0 PL=0
MOVL C01215 V=800.0 PL=0
MOVL C01216 V=800.0 PL=0
MOVL C01217 V=800.0 PL=0
MOVL C01218 V=800.0 PL=0
MOVL C01219 V=800.0 PL=0
MOVL C01220 V=800.0 PL=0
MOVL C01221 V=800.0 PL=0
MOVL C01222 V=800.0 PL=0
MOVL C01223 V=800.0 PL=0
MOVL C01224 V=800.0 PL=0
MOVL C01225 V=800.0 PL=0
MOVL C01226 V=800.0 PL=0
MOVL C01227 V=800.0 PL=0
MOVL C01228 V=800.0 PL=0
MOVL C01229 V=800.0 PL=0
MOVL C01230 V=800.0 PL=0
MOVL C01231 V=800.0 PL=0
MOVL C01232 V=800.0 PL=0
MOVL C01233 V=800.0 PL=0
MOVL C01234 V=800.0 PL=0
MOVL C01235 V=800.0 PL=0
MOVL C01236 V=800.0 PL=0
MOVL C01237 V=800.0 PL=0
MOVL C01238 V=800.0 PL=0
MOVL C01239 V=800.0 PL=0
MOVL C01240 V=800.0 PL=0
MOVL C01241 V=800.0 PL=0
MOVL C01242 V=800.0 PL=0
MOVL C01243 V=800.0 PL=0
MOVL C01244 V=800.0 PL=0
MOVL C01245 V=800.0 PL=0
MOVL C01246 V=800.0 PL=0
MOVL C01247 V=800.0 PL=0
MOVL C01248 V=800.0 PL=0
MOVL C01249 V=800.0 PL=0
MOVL C01250 V=800.0 PL=0
MOVL C01251 V=800.0 PL=0
MOVL C01252 V=800.0 PL=0
MOVL C01253 V=800.0 PL=0
MOVL C01254 V=800.0 PL=0
MOVL C01255 V=800.0 PL=0
MOVL C01256 V=800.0 PL=0
MOVL C01257 V=800.0 PL=0
MOVL C01258 V=800.0 PL=0
MOVL C01259 V=800.0 PL=0
MOVL C01260 V=800.0 PL=0
MOVL C01261 V=800.0 PL=0
MOVL C01262 V=800.0 PL=0
MOVL C01263 V=800.0 PL=0
MOVL C01264 V=800.0 PL=0
MOVL C01265 V=800.0 PL=0
MOVL C01266 V=800.0 PL=0
MOVL C01267 V=800.0 PL=0
MOVL C01268 V=800.0 PL=0
MOVL C01269 V=800.0 PL=0
MOVL C01270 V=800.0 PL=0
MOVL C01271 V=800.0 PL=0
MOVL C01272 V=800.0 PL=0
MOVL C01273 V=800.0 PL=0
MOVL C01274 V=800.0 PL=0
MOVL C01275 V=800.0 PL=0
MOVL C01276 V=800.0 PL=0
MOVL C01277 V=800.0 PL=0
MOVL C01278 V=800.0 PL=0
MOVL C01279 V=800.0 PL=0
MOVL C01280 V=800.0 PL=0
MOVL C01281 V=800.0 PL=0
MOVL C01282 V=800.0 PL=0
MOVL C01283 V=800.0 PL=0
MOVL C01284 V=800.0 PL=0
MOVL C01285 V=800.0 PL=0
MOVL C01286 V=800.0 PL=0
MOVL C01287 V=800.0 PL=0
MOVL C01288 V=800.0 PL=0
MOVL C01289 V=800.0 PL=0
MOVL C01290 V=800.0 PL=0
MOVL C01291 V=800.0 PL=0
MOVL C01292 V=800.0 PL=0
MOVL C01293 V=800.0 PL=0
MOVL C01294 V=800.0 PL=0
MOVL C01295 V=800.0 PL=0
MOVL C01296 V=800.0 PL=0
MOVL C01297 V=800.0 PL=0
MOVL C01298 V=800.0 PL=0
MOVL C01299 V=800.0 PL=0
MOVL C01300 V=800.0 PL=0
MOVL C01301 V=800.0 PL=0
MOVL C01302 V=800.0 PL=0
MOVL C01303 V=800.0 PL=0
MOVL C01304 V=800.0 PL=0
MOVL C01305 V=800.0 PL=0
MOVL C01306 V=800.0 PL=0
MOVL C01307 V=800.0 PL=0
MOVL C01308 V=800.0 PL=0
MOVL C01309 V=800.0 PL=0
MOVL C01310 V=800.0 PL=0
MOVL C01311 V=800.0 PL=0
MOVL C01312 V=800.0 PL=0
MOVL C01313 V=800.0 PL=0
MOVL C01314 V=800.0 PL=0
MOVL C01315 V=800.0 PL=0
MOVL C01316 V=800.0 PL=0
MOVL C01317 V=800.0 PL=0
MOVL C01318 V=800.0 PL=0
MOVL C01319 V=800.0 PL=0
MOVL C01320 V=800.0 PL=0
MOVL C01321 V=800.0 PL=0
MOVL C01322 V=800.0 PL=0
MOVL C01323 V=800.0 PL=0
MOVL C01324 V=800.0 PL=0
MOVL C01325 V=800.0 PL=0
MOVL C01326 V=800.0 PL=0
MOVL C01327 V=800.0 PL=0
MOVL C01328 V=800.0 PL=0
MOVL C01329 V=800.0 PL=0
MOVL C01330 V=800.0 PL=0
MOVL C01331 V=800.0 PL=0
MOVL C01332 V=800.0 PL=0
MOVL C01333 V=800.0 PL=0
MOVL C01334 V=800.0 PL=0
MOVL C01335 V=800.0 PL=0
MOVL C01336 V=800.0 PL=0
MOVL C01337 V=800.0 PL=0
MOVL C01338 V=800.0 PL=0
MOVL C01339 V=800.0 PL=0
MOVL C01340 V=800.0 PL=0
MOVL C01341 V=800.0 PL=0
MOVL C01342 V=800.0 PL=0
MOVL C01343 V=800.0 PL=0
MOVL C01344 V=800.0 PL=0
MOVL C01345 V=800.0 PL=0
MOVL C01346 V=800.0 PL=0
MOVL C01347 V=800.0 PL=0
MOVL C01348 V=800.0 PL=0
MOVL C01349 V=800.0 PL=0
MOVL C01350 V=800.0 PL=0
MOVL C01351 V=800.0 PL=0
MOVL C01352 V=800.0 PL=0
MOVL C01353 V=800.0 PL=0
MOVL C01354 V=800.0 PL=0
MOVL C01355 V=800.0 PL=0
MOVL C01356 V=800.0 PL=0
MOVL C01357 V=800.0 PL=0
MOVL C01358 V=800.0 PL=0
MOVL C01359 V=800.0 PL=0
MOVL C01360 V=800.0 PL=0
MOVL C01361 V=800.0 PL=0
MOVL C01362 V=800.0 PL=0
MOVL C01363 V=800.0 PL=0
MOVL C01364 V=800.0 PL=0
MOVL C01365 V=800.0 PL=0
MOVL C01366 V=800.0 PL=0
MOVL C01367 V=800.0 PL=0
MOVL C01368 V=800.0 PL=0
MOVL C01369 V=800.0 PL=0
MOVL C01370 V=800.0 PL=0
MOVL C01371 V=800.0 PL=0
MOVL C01372 V=800.0 PL=0
MOVL C01373 V=800.0 PL=0
MOVL C01374 V=800.0 PL=0
MOVL C01375 V=800.0 PL=0
MOVL C01376 V=800.0 PL=0
MOVL C01377 V=800.0 PL=0
MOVL C01378 V=800.0 PL=0
MOVL C01379 V=800.0 PL=0
MOVL C01380 V=800.0 PL=0
MOVL C01381 V=800.0 PL=0
MOVL C01382 V=800.0 PL=0
MOVL C01383 V=800.0 PL=0
MOVL C01384 V=800.0 PL=0
MOVL C01385 V=800.0 PL=0
MOVL C01386 V=800.0 PL=0
MOVL C01387 V=800.0 PL=0
MOVL C01388 V=800.0 PL=0
MOVL C01389 V=800.0 PL=0
MOVL C01390 V=800.0 PL=0
MOVL C01391 V=800.0 PL=0
MOVL C01392 V=800.0 PL=0
MOVL C01393 V=800.0 PL=0
MOVL C01394 V=800.0 PL=0
MOVL C01395 V=800.0 PL=0
MOVL C01396 V=800.0 PL=0
MOVL C01397 V=800.0 PL=0
MOVL C01398 V=800.0 PL=0
MOVL C01399 V=800.0 PL=0
MOVL C01400 V=800.0 PL=0
MOVL C01401 V=800.0 PL=0
MOVL C01402 V=800.0 PL=0
MOVL C01403 V=800.0 PL=0
MOVL C01404 V=800.0 PL=0
MOVL C01405 V=800.0 PL=0
MOVL C01406 V=800.0 PL=0
MOVL C01407 V=800.0 PL=0
MOVL C01408 V=800.0 PL=0
MOVL C01409 V=800.0 PL=0
MOVL C01410 V=800.0 PL=0
MOVL C01411 V=800.0 PL=0
MOVL C01412 V=800.0 PL=0
MOVL C01413 V=800.0 PL=0
MOVL C01414 V=800.0 PL=0
MOVL C01415 V=800.0 PL=0
MOVL C01416 V=800.0 PL=0
MOVL C01417 V=800.0 PL=0
MOVL C01418 V=800.0 PL=0
MOVL C01419 V=800.0 PL=0
MOVL C01420 V=800.0 PL=0
MOVL C01421 V=800.0 PL=0
MOVL C01422 V=800.0 PL=0
MOVL C01423 V=800.0 PL=0
MOVL C01424 V=800.0 PL=0
MOVL C01425 V=800.0 PL=0
MOVL C01426 V=800.0 PL=0
MOVL C01427 V=800.0 PL=0
MOVL C01428 V=800.0 PL=0
MOVL C01429 V=800.0 PL=0
MOVL C01430 V=800.0 PL=0
MOVL C01431 V=800.0 PL=0
MOVL C01432 V=800.0 PL=0
MOVL C01433 V=800.0 PL=0
MOVL C01434 V=800.0 PL=0
MOVL C01435 V=800.0 PL=0
MOVL C01436 V=800.0 PL=0
MOVL C01437 V=800.0 PL=0
MOVL C01438 V=800.0 PL=0
MOVL C01439 V=800.0 PL=0
MOVL C01440 V=800.0 PL=0
MOVL C01441 V=800.0 PL=0
MOVL C01442 V=800.0 PL=0
MOVL C01443 V=800.0 PL=0
MOVL C01444 V=800.0 PL=0
MOVL C01445 V=800.0 PL=0
MOVL C01446 V=800.0 PL=0
MOVL C01447 V=800.0 PL=0
MOVL C01448 V=800.0 PL=0
MOVL C01449 V=800.0 PL=0
MOVL C01450 V=800.0 PL=0
MOVL C01451 V=800.0 PL=0
MOVL C01452 V=800.0 PL=0
MOVL C01453 V=800.0 PL=0
MOVL C01454 V=800.0 PL=0
MOVL C01455 V=800.0 PL=0
MOVL C01456 V=800.0 PL=0
MOVL C01457 V=800.0 PL=0
MOVL C01458 V=800.0 PL=0
MOVL C01459 V=800.0 PL=0
MOVL C01460 V=800.0 PL=0
MOVL C01461 V=800.0 PL=0
MOVL C01462 V=800.0 PL=0
MOVL C01463 V=800.0 PL=0
MOVL C01464 V=800.0 PL=0
MOVL C01465 V=800.0 PL=0
MOVL C01466 V=800.0 PL=0
MOVL C01467 V=800.0 PL=0
MOVL C01468 V=800.0 PL=0
MOVL C01469 V=800.0 PL=0
MOVL C01470 V=800.0 PL=0
MOVL C01471 V=800.0 PL=0
MOVL C01472 V=800.0 PL=0
MOVL C01473 V=800.0 PL=0
MOVL C01474 V=800.0 PL=0
MOVL C01475 V=800.0 PL=0
MOVL C01476 V=800.0 PL=0
MOVL C01477 V=800.0 PL=0
MOVL C01478 V=800.0 PL=0
MOVL C01479 V=800.0 PL=0
MOVL C01480 V=800.0 PL=0
MOVL C01481 V=800.0 PL=0
MOVL C01482 V=800.0 PL=0
MOVL C01483 V=800.0 PL=0
MOVL C01484 V=800.0 PL=0
MOVL C01485 V=800.0 PL=0
MOVL C01486 V=800.0 PL=0
MOVL C01487 V=800.0 PL=0
MOVL C01488 V=800.0 PL=0
MOVL C01489 V=800.0 PL=0
MOVL C01490 V=800.0 PL=0
MOVL C01491 V=800.0 PL=0
MOVL C01492 V=800.0 PL=0
MOVL C01493 V=800.0 PL=0
MOVL C01494 V=800.0 PL=0
MOVL C01495 V=800.0 PL=0
MOVL C01496 V=800.0 PL=0
MOVL C01497 V=800.0 PL=0
MOVL C01498 V=800.0 PL=0
MOVL C01499 V=800.0 PL=0
MOVL C01500 V=800.0 PL=0
MOVL C01501 V=800.0 PL=0
MOVL C01502 V=800.0 PL=0
MOVL C01503 V=800.0 PL=0
MOVL C01504 V=800.0 PL=0
MOVL C01505 V=800.0 PL=0
MOVL C01506 V=800.0 PL=0
MOVL C01507 V=800.0 PL=0
MOVL C01508 V=800.0 PL=0
MOVL C01509 V=800.0 PL=0
MOVL C01510 V=800.0 PL=0
MOVL C01511 V=800.0 PL=0
MOVL C01512 V=800.0 PL=0
MOVL C01513 V=800.0 PL=0
MOVL C01514 V=800.0 PL=0
MOVL C01515 V=800.0 PL=0
MOVL C01516 V=800.0 PL=0
MOVL C01517 V=800.0 PL=0
MOVL C01518 V=800.0 PL=0
MOVL C01519 V=800.0 PL=0
MOVL C01520 V=800.0 PL=0
MOVL C01521 V=800.0 PL=0
MOVL C01522 V=800.0 PL=0
MOVL C01523 V=800.0 PL=0
MOVL C01524 V=800.0 PL=0
MOVL C01525 V=800.0 PL=0
MOVL C01526 V=800.0 PL=0
MOVL C01527 V=800.0 PL=0
MOVL C01528 V=800.0 PL=0
MOVL C01529 V=800.0 PL=0
MOVL C01530 V=800.0 PL=0
MOVL C01531 V=800.0 PL=0
MOVL C01532 V=800.0 PL=0
MOVL C01533 V=800.0 PL=0
MOVL C01534 V=800.0 PL=0
MOVL C01535 V=800.0 PL=0
MOVL C01536 V=800.0 PL=0
MOVL C01537 V=800.0 PL=0
MOVL C01538 V=800.0 PL=0
MOVL C01539 V=800.0 PL=0
MOVL C01540 V=800.0 PL=0
MOVL C01541 V=800.0 PL=0
MOVL C01542 V=800.0 PL=0
MOVL C01543 V=800.0 PL=0
MOVL C01544 V=800.0 PL=0
MOVL C01545 V=800.0 PL=0
MOVL C01546 V=800.0 PL=0
MOVL C01547 V=800.0 PL=0
MOVL C01548 V=800.0 PL=0
MOVL C01549 V=800.0 PL=0
MOVL C01550 V=800.0 PL=0
MOVL C01551 V=800.0 PL=0
MOVL C01552 V=800.0 PL=0
MOVL C01553 V=800.0 PL=0
MOVL C01554 V=800.0 PL=0
MOVL C01555 V=800.0 PL=0
MOVL C01556 V=800.0 PL=0
MOVL C01557 V=800.0 PL=0
MOVL C01558 V=800.0 PL=0
MOVL C01559 V=800.0 PL=0
MOVL C01560 V=800.0 PL=0
MOVL C01561 V=800.0 PL=0
MOVL C01562 V=800.0 PL=0
MOVL C01563 V=800.0 PL=0
MOVL C01564 V=800.0 PL=0
MOVL C01565 V=800.0 PL=0
MOVL C01566 V=800.0 PL=0
MOVL C01567 V=800.0 PL=0
MOVL C01568 V=800.0 PL=0
MOVL C01569 V=800.0 PL=0
MOVL C01570 V=800.0 PL=0
MOVL C01571 V=800.0 PL=0
MOVL C01572 V=800.0 PL=0
MOVL C01573 V=800.0 PL=0
MOVL C01574 V=800.0 PL=0
MOVL C01575 V=800.0 PL=0
MOVL C01576 V=800.0 PL=0
MOVL C01577 V=800.0 PL=0
MOVL C01578 V=800.0 PL=0
MOVL C01579 V=800.0 PL=0
MOVL C01580 V=800.0 PL=0
MOVL C01581 V=800.0 PL=0
MOVL C01582 V=800.0 PL=0
MOVL C01583 V=800.0 PL=0
MOVL C01584 V=800.0 PL=0
MOVL C01585 V=800.0 PL=0
MOVL C01586 V=800.0 PL=0
MOVL C01587 V=800.0 PL=0
MOVL C01588 V=800.0 PL=0
MOVL C01589 V=800.0 PL=0
MOVL C01590 V=800.0 PL=0
MOVL C01591 V=800.0 PL=0
MOVL C01592 V=800.0 PL=0
MOVL C01593 V=800.0 PL=0
MOVL C01594 V=800.0 PL=0
MOVL C01595 V=800.0 PL=0
MOVL C01596 V=800.0 PL=0
MOVL C01597 V=800.0 PL=0
MOVL C01598 V=800.0 PL=0
MOVL C01599 V=800.0 PL=0
MOVL C01600 V=800.0 PL=0
MOVL C01601 V=800.0 PL=0
MOVL C01602 V=800.0 PL=0
MOVL C01603 V=800.0 PL=0
MOVL C01604 V=800.0 PL=0
MOVL C01605 V=800.0 PL=0
MOVL C01606 V=800.0 PL=0
MOVL C01607 V=800.0 PL=0
MOVL C01608 V=800.0 PL=0
MOVL C01609 V=800.0 PL=0
MOVL C01610 V=800.0 PL=0
MOVL C01611 V=800.0 PL=0
MOVL C01612 V=800.0 PL=0
MOVL C01613 V=800.0 PL=0
MOVL C01614 V=800.0 PL=0
MOVL C01615 V=800.0 PL=0
MOVL C01616 V=800.0 PL=0
MOVL C01617 V=800.0 PL=0
MOVL C01618 V=800.0 PL=0
MOVL C01619 V=800.0 PL=0
MOVL C01620 V=800.0 PL=0
MOVL C01621 V=800.0 PL=0
MOVL C01622 V=800.0 PL=0
MOVL C01623 V=800.0 PL=0
MOVL C01624 V=800.0 PL=0
MOVL C01625 V=800.0 PL=0
MOVL C01626 V=800.0 PL=0
MOVL C01627 V=800.0 PL=0
MOVL C01628 V=800.0 PL=0
MOVL C01629 V=800.0 PL=0
MOVL C01630 V=800.0 PL=0
MOVL C01631 V=800.0 PL=0
MOVL C01632 V=800.0 PL=0
MOVL C01633 V=800.0 PL=0
MOVL C01634 V=800.0 PL=0
MOVL C01635 V=800.0 PL=0
MOVL C01636 V=800.0 PL=0
MOVL C01637 V=800.0 PL=0
MOVL C01638 V=800.0 PL=0
MOVL C01639 V=800.0 PL=0
MOVL C01640 V=800.0 PL=0
MOVL C01641 V=800.0 PL=0
MOVL C01642 V=800.0 PL=0
MOVL C01643 V=800.0 PL=0
MOVL C01644 V=800.0 PL=0
MOVL C01645 V=800.0 PL=0
MOVL C01646 V=800.0 PL=0
MOVL C01647 V=800.0 PL=0
MOVL C01648 V=800.0 PL=0
MOVL C01649 V=800.0 PL=0
MOVL C01650 V=800.0 PL=0
MOVL C01651 V=800.0 PL=0
MOVL C01652 V=800.0 PL=0
MOVL C01653 V=800.0 PL=0
MOVL C01654 V=800.0 PL=0
MOVL C01655 V=800.0 PL=0
MOVL C01656 V=800.0 PL=0
MOVL C01657 V=800.0 PL=0
MOVL C01658 V=800.0 PL=0
MOVL C01659 V=800.0 PL=0
MOVL C01660 V=800.0 PL=0
MOVL C01661 V=800.0 PL=0
MOVL C01662 V=800.0 PL=0
MOVL C01663 V=800.0 PL=0
MOVL C01664 V=800.0 PL=0
MOVL C01665 V=800.0 PL=0
MOVL C01666 V=800.0 PL=0
MOVL C01667 V=800.0 PL=0
MOVL C01668 V=800.0 PL=0
MOVL C01669 V=800.0 PL=0
MOVL C01670 V=800.0 PL=0
MOVL C01671 V=800.0 PL=0
MOVL C01672 V=800.0 PL=0
MOVL C01673 V=800.0 PL=0
MOVL C01674 V=800.0 PL=0
MOVL C01675 V=800.0 PL=0
MOVL C01676 V=800.0 PL=0
MOVL C01677 V=800.0 PL=0
MOVL C01678 V=800.0 PL=0
MOVL C01679 V=800.0 PL=0
MOVL C01680 V=800.0 PL=0
MOVL C01681 V=800.0 PL=0
MOVL C01682 V=800.0 PL=0
MOVL C01683 V=800.0 PL=0
MOVL C01684 V=800.0 PL=0
MOVL C01685 V=800.0 PL=0
MOVL C01686 V=800.0 PL=0
MOVL C01687 V=800.0 PL=0
MOVL C01688 V=800.0 PL=0
MOVL C01689 V=800.0 PL=0
MOVL C01690 V=800.0 PL=0
MOVL C01691 V=800.0 PL=0
MOVL C01692 V=800.0 PL=0
MOVL C01693 V=800.0 PL=0
MOVL C01694 V=800.0 PL=0
MOVL C01695 V=800.0 PL=0
MOVL C01696 V=800.0 PL=0
MOVL C01697 V=800.0 PL=0
MOVL C01698 V=800.0 PL=0
MOVL C01699 V=800.0 PL=0
MOVL C01700 V=800.0 PL=0
MOVL C01701 V=800.0 PL=0
MOVL C01702 V=800.0 PL=0
MOVL C01703 V=800.0 PL=0
MOVL C01704 V=800.0 PL=0
MOVL C01705 V=800.0 PL=0
MOVL C01706 V=800.0 PL=0
MOVL C01707 V=800.0 PL=0
MOVL C01708 V=800.0 PL=0
MOVL C01709 V=800.0 PL=0
MOVL C01710 V=800.0 PL=0
MOVL C01711 V=800.0 PL=0
MOVL C01712 V=800.0 PL=0
MOVL C01713 V=800.0 PL=0
MOVL C01714 V=800.0 PL=0
MOVL C01715 V=800.0 PL=0
MOVL C01716 V=800.0 PL=0
MOVL C01717 V=800.0 PL=0
MOVL C01718 V=800.0 PL=0
MOVL C01719 V=800.0 PL=0
MOVL C01720 V=800.0 PL=0
MOVL C01721 V=800.0 PL=0
MOVL C01722 V=800.0 PL=0
MOVL C01723 V=800.0 PL=0
MOVL C01724 V=800.0 PL=0
MOVL C01725 V=800.0 PL=0
MOVL C01726 V=800.0 PL=0
MOVL C01727 V=800.0 PL=0
MOVL C01728 V=800.0 PL=0
MOVL C01729 V=800.0 PL=0
MOVL C01730 V=800.0 PL=0
MOVL C01731 V=800.0 PL=0
MOVL C01732 V=800.0 PL=0
MOVL C01733 V=800.0 PL=0
MOVL C01734 V=800.0 PL=0
MOVL C01735 V=800.0 PL=0
MOVL C01736 V=800.0 PL=0
MOVL C01737 V=800.0 PL=0
MOVL C01738 V=800.0 PL=0
MOVL C01739 V=800.0 PL=0
MOVL C01740 V=800.0 PL=0
MOVL C01741 V=800.0 PL=0
MOVL C01742 V=800.0 PL=0
MOVL C01743 V=800.0 PL=0
MOVL C01744 V=800.0 PL=0
MOVL C01745 V=800.0 PL=0
MOVL C01746 V=800.0 PL=0
MOVL C01747 V=800.0 PL=0
MOVL C01748 V=800.0 PL=0
MOVL C01749 V=800.0 PL=0
MOVL C01750 V=800.0 PL=0
MOVL C01751 V=800.0 PL=0
MOVL C01752 V=800.0 PL=0
MOVL C01753 V=800.0 PL=0
MOVL C01754 V=800.0 PL=0
MOVL C01755 V=800.0 PL=0
MOVL C01756 V=800.0 PL=0
MOVL C01757 V=800.0 PL=0
MOVL C01758 V=800.0 PL=0
MOVL C01759 V=800.0 PL=0
MOVL C01760 V=800.0 PL=0
MOVL C01761 V=800.0 PL=0
MOVL C01762 V=800.0 PL=0
MOVL C01763 V=800.0 PL=0
MOVL C01764 V=800.0 PL=0
MOVL C01765 V=800.0 PL=0
MOVL C01766 V=800.0 PL=0
MOVL C01767 V=800.0 PL=0
MOVL C01768 V=800.0 PL=0
MOVL C01769 V=800.0 PL=0
MOVL C01770 V=800.0 PL=0
MOVL C01771 V=800.0 PL=0
MOVL C01772 V=800.0 PL=0
MOVL C01773 V=800.0 PL=0
MOVL C01774 V=800.0 PL=0
MOVL C01775 V=800.0 PL=0
MOVL C01776 V=800.0 PL=0
MOVL C01777 V=800.0 PL=0
MOVL C01778 V=800.0 PL=0
MOVL C01779 V=800.0 PL=0
MOVL C01780 V=800.0 PL=0
MOVL C01781 V=800.0 PL=0
MOVL C01782 V=800.0 PL=0
MOVL C01783 V=800.0 PL=0
MOVL C01784 V=800.0 PL=0
MOVL C01785 V=800.0 PL=0
MOVL C01786 V=800.0 PL=0
MOVL C01787 V=800.0 PL=0
MOVL C01788 V=800.0 PL=0
MOVL C01789 V=800.0 PL=0
MOVL C01790 V=800.0 PL=0
MOVL C01791 V=800.0 PL=0
MOVL C01792 V=800.0 PL=0
MOVL C01793 V=800.0 PL=0
MOVL C01794 V=800.0 PL=0
MOVL C01795 V=800.0 PL=0
MOVL C01796 V=800.0 PL=0
MOVL C01797 V=800.0 PL=0
MOVL C01798 V=800.0 PL=0
MOVL C01799 V=800.0 PL=0
MOVL C01800 V=800.0 PL=0
MOVL C01801 V=800.0 PL=0
MOVL C01802 V=800.0 PL=0
MOVL C01803 V=800.0 PL=0
MOVL C01804 V=800.0 PL=0
MOVL C01805 V=800.0 PL=0
MOVL C01806 V=800.0 PL=0
MOVL C01807 V=800.0 PL=0
MOVL C01808 V=800.0 PL=0
MOVL C01809 V=800.0 PL=0
MOVL C01810 V=800.0 PL=0
MOVL C01811 V=800.0 PL=0
MOVL C01812 V=800.0 PL=0
MOVL C01813 V=800.0 PL=0
MOVL C01814 V=800.0 PL=0
MOVL C01815 V=800.0 PL=0
MOVL C01816 V=800.0 PL=0
MOVL C01817 V=800.0 PL=0
MOVL C01818 V=800.0 PL=0
MOVL C01819 V=800.0 PL=0
MOVL C01820 V=800.0 PL=0
MOVL C01821 V=800.0 PL=0
MOVL C01822 V=800.0 PL=0
MOVL C01823 V=800.0 PL=0
MOVL C01824 V=800.0 PL=0
MOVL C01825 V=800.0 PL=0
MOVL C01826 V=800.0 PL=0
MOVL C01827 V=800.0 PL=0
MOVL C01828 V=800.0 PL=0
MOVL C01829 V=800.0 PL=0
MOVL C01830 V=800.0 PL=0
MOVL C01831 V=800.0 PL=0
MOVL C01832 V=800.0 PL=0
MOVL C01833 V=800.0 PL=0
MOVL C01834 V=800.0 PL=0
MOVL C01835 V=800.0 PL=0
MOVL C01836 V=800.0 PL=0
MOVL C01837 V=800.0 PL=0
MOVL C01838 V=800.0 PL=0
MOVL C01839 V=800.0 PL=0
MOVL C01840 V=800.0 PL=0
MOVL C01841 V=800.0 PL=0
MOVL C01842 V=800.0 PL=0
MOVL C01843 V=800.0 PL=0
MOVL C01844 V=800.0 PL=0
MOVL C01845 V=800.0 PL=0
MOVL C01846 V=800.0 PL=0
MOVL C01847 V=800.0 PL=0
MOVL C01848 V=800.0 PL=0
MOVL C01849 V=800.0 PL=0
MOVL C01850 V=800.0 PL=0
MOVL C01851 V=800.0 PL=0
MOVL C01852 V=800.0 PL=0
MOVL C01853 V=800.0 PL=0
MOVL C01854 V=800.0 PL=0
MOVL C01855 V=800.0 PL=0
MOVL C01856 V=800.0 PL=0
MOVL C01857 V=800.0 PL=0
MOVL C01858 V=800.0 PL=0
MOVL C01859 V=800.0 PL=0
MOVL C01860 V=800.0 PL=0
MOVL C01861 V=800.0 PL=0
MOVL C01862 V=800.0 PL=0
MOVL C01863 V=800.0 PL=0
MOVL C01864 V=800.0 PL=0
MOVL C01865 V=800.0 PL=0
MOVL C01866 V=800.0 PL=0
MOVL C01867 V=800.0 PL=0
MOVL C01868 V=800.0 PL=0
MOVL C01869 V=800.0 PL=0
MOVL C01870 V=800.0 PL=0
MOVL C01871 V=800.0 PL=0
MOVL C01872 V=800.0 PL=0
MOVL C01873 V=800.0 PL=0
MOVL C01874 V=800.0 PL=0
MOVL C01875 V=800.0 PL=0
MOVL C01876 V=800.0 PL=0
MOVL C01877 V=800.0 PL=0
MOVL C01878 V=800.0 PL=0
MOVL C01879 V=800.0 PL=0
MOVL C01880 V=800.0 PL=0
MOVL C01881 V=800.0 PL=0
MOVL C01882 V=800.0 PL=0
MOVL C01883 V=800.0 PL=0
MOVL C01884 V=800.0 PL=0
MOVL C01885 V=800.0 PL=0
MOVL C01886 V=800.0 PL=0
MOVL C01887 V=800.0 PL=0
MOVL C01888 V=800.0 PL=0
MOVL C01889 V=800.0 PL=0
MOVL C01890 V=800.0 PL=0
MOVL C01891 V=800.0 PL=0
MOVL C01892 V=800.0 PL=0
MOVL C01893 V=800.0 PL=0
MOVL C01894 V=800.0 PL=0
MOVL C01895 V=800.0 PL=0
MOVL C01896 V=800.0 PL=0
MOVL C01897 V=800.0 PL=0
MOVL C01898 V=800.0 PL=0
MOVL C01899 V=800.0 PL=0
MOVL C01900 V=800.0 PL=0
MOVL C01901 V=800.0 PL=0
MOVL C01902 V=800.0 PL=0
MOVL C01903 V=800.0 PL=0
MOVL C01904 V=800.0 PL=0
MOVL C01905 V=800.0 PL=0
MOVL C01906 V=800.0 PL=0
MOVL C01907 V=800.0 PL=0
MOVL C01908 V=800.0 PL=0
MOVL C01909 V=800.0 PL=0
MOVL C01910 V=800.0 PL=0
MOVL C01911 V=800.0 PL=0
MOVL C01912 V=800.0 PL=0
MOVL C01913 V=800.0 PL=0
MOVL C01914 V=800.0 PL=0
MOVL C01915 V=800.0 PL=0
MOVL C01916 V=800.0 PL=0
MOVL C01917 V=800.0 PL=0
MOVL C01918 V=800.0 PL=0
MOVL C01919 V=800.0 PL=0
MOVL C01920 V=800.0 PL=0
MOVL C01921 V=800.0 PL=0
MOVL C01922 V=800.0 PL=0
MOVL C01923 V=800.0 PL=0
MOVL C01924 V=800.0 PL=0
MOVL C01925 V=800.0 PL=0
MOVL C01926 V=800.0 PL=0
MOVL C01927 V=800.0 PL=0
MOVL C01928 V=800.0 PL=0
MOVL C01929 V=800.0 PL=0
MOVL C01930 V=800.0 PL=0
MOVL C01931 V=800.0 PL=0
MOVL C01932 V=800.0 PL=0
MOVL C01933 V=800.0 PL=0
MOVL C01934 V=800.0 PL=0
MOVL C01935 V=800.0 PL=0
MOVL C01936 V=800.0 PL=0
MOVL C01937 V=800.0 PL=0
MOVL C01938 V=800.0 PL=0
MOVL C01939 V=800.0 PL=0
MOVL C01940 V=800.0 PL=0
MOVL C01941 V=800.0 PL=0
MOVL C01942 V=800.0 PL=0
MOVL C01943 V=800.0 PL=0
MOVL C01944 V=800.0 PL=0
MOVL C01945 V=800.0 PL=0
MOVL C01946 V=800.0 PL=0
MOVL C01947 V=800.0 PL=0
MOVL C01948 V=800.0 PL=0
MOVL C01949 V=800.0 PL=0
MOVL C01950 V=800.0 PL=0
MOVL C01951 V=800.0 PL=0
MOVL C01952 V=800.0 PL=0
MOVL C01953 V=800.0 PL=0
MOVL C01954 V=800.0 PL=0
MOVL C01955 V=800.0 PL=0
MOVL C01956 V=800.0 PL=0
MOVL C01957 V=800.0 PL=0
MOVL C01958 V=800.0 PL=0
MOVL C01959 V=800.0 PL=0
MOVL C01960 V=800.0 PL=0
MOVL C01961 V=800.0 PL=0
MOVL C01962 V=800.0 PL=0
MOVL C01963 V=800.0 PL=0
MOVL C01964 V=800.0 PL=0
MOVL C01965 V=800.0 PL=0
MOVL C01966 V=800.0 PL=0
MOVL C01967 V=800.0 PL=0
MOVL C01968 V=800.0 PL=0
MOVL C01969 V=800.0 PL=0
MOVL C01970 V=800.0 PL=0
MOVL C01971 V=800.0 PL=0
MOVL C01972 V=800.0 PL=0
MOVL C01973 V=800.0 PL=0
MOVL C01974 V=800.0 PL=0
MOVL C01975 V=800.0 PL=0
MOVL C01976 V=800.0 PL=0
MOVL C01977 V=800.0 PL=0
MOVL C01978 V=800.0 PL=0
MOVL C01979 V=800.0 PL=0
MOVL C01980 V=800.0 PL=0
MOVL C01981 V=800.0 PL=0
MOVL C01982 V=800.0 PL=0
MOVL C01983 V=800.0 PL=0
MOVL C01984 V=800.0 PL=0
MOVL C01985 V=800.0 PL=0
MOVL C01986 V=800.0 PL=0
MOVL C01987 V=800.0 PL=0
MOVL C01988 V=800.0 PL=0
MOVL C01989 V=800.0 PL=0
MOVL C01990 V=800.0 PL=0
MOVL C01991 V=800.0 PL=0
MOVL C01992 V=800.0 PL=0
MOVL C01993 V=800.0 PL=0
MOVL C01994 V=800.0 PL=0
MOVL C01995 V=800.0 PL=0
MOVL C01996 V=800.0 PL=0
MOVL C01997 V=800.0 PL=0
MOVL C01998 V=800.0 PL=0
MOVL C01999 V=800.0 PL=0
MOVL C02000 V=800.0 PL=0
MOVL C02001 V=800.0 PL=0
MOVL C02002 V=800.0 PL=0
MOVL C02003 V=800.0 PL=0
MOVL C02004 V=800.0 PL=0
MOVL C02005 V=800.0 PL=0
MOVL C02006 V=800.0 PL=0
MOVL C02007 V=800.0 PL=0
MOVL C02008 V=800.0 PL=0
MOVL C02009 V=800.0 PL=0
MOVL C02010 V=800.0 PL=0
MOVL C02011 V=800.0 PL=0
MOVL C02012 V=800.0 PL=0
MOVL C02013 V=800.0 PL=0
MOVL C02014 V=800.0 PL=0
MOVL C02015 V=800.0 PL=0
MOVL C02016 V=800.0 PL=0
MOVL C02017 V=800.0 PL=0
MOVL C02018 V=800.0 PL=0
MOVL C02019 V=800.0 PL=0
MOVL C02020 V=800.0 PL=0
MOVL C02021 V=800.0 PL=0
MOVL C02022 V=800.0 PL=0
MOVL C02023 V=800.0 PL=0
MOVL C02024 V=800.0 PL=0
MOVL C02025 V=800.0 PL=0
MOVL C02026 V=800.0 PL=0
MOVL C02027 V=800.0 PL=0
MOVL C02028 V=800.0 PL=0
MOVL C02029 V=800.0 PL=0
MOVL C02030 V=800.0 PL=0
MOVL C02031 V=800.0 PL=0
MOVL C02032 V=800.0 PL=0
MOVL C02033 V=800.0 PL=0
MOVL C02034 V=800.0 PL=0
MOVL C02035 V=800.0 PL=0
MOVL C02036 V=800.0 PL=0
MOVL C02037 V=800.0 PL=0
MOVL C02038 V=800.0 PL=0
MOVL C02039 V=800.0 PL=0
MOVL C02040 V=800.0 PL=0
MOVL C02041 V=800.0 PL=0
MOVL C02042 V=800.0 PL=0
MOVL C02043 V=800.0 PL=0
MOVL C02044 V=800.0 PL=0
MOVL C02045 V=800.0 PL=0
MOVL C02046 V=800.0 PL=0
MOVL C02047 V=800.0 PL=0
MOVL C02048 V=800.0 PL=0
MOVL C02049 V=800.0 PL=0
MOVL C02050 V=800.0 PL=0
MOVL C02051 V=800.0 PL=0
MOVL C02052 V=800.0 PL=0
MOVL C02053 V=800.0 PL=0
MOVL C02054 V=800.0 PL=0
MOVL C02055 V=800.0 PL=0
MOVL C02056 V=800.0 PL=0
MOVL C02057 V=800.0 PL=0
MOVL C02058 V=800.0 PL=0
MOVL C02059 V=800.0 PL=0
MOVL C02060 V=800.0 PL=0
MOVL C02061 V=800.0 PL=0
MOVL C02062 V=800.0 PL=0
MOVL C02063 V=800.0 PL=0
MOVL C02064 V=800.0 PL=0
MOVL C02065 V=800.0 PL=0
MOVL C02066 V=800.0 PL=0
MOVL C02067 V=800.0 PL=0
MOVL C02068 V=800.0 PL=0
MOVL C02069 V=800.0 PL=0
MOVL C02070 V=800.0 PL=0
MOVL C02071 V=800.0 PL=0
MOVL C02072 V=800.0 PL=0
MOVL C02073 V=800.0 PL=0
MOVL C02074 V=800.0 PL=0
MOVL C02075 V=800.0 PL=0
MOVL C02076 V=800.0 PL=0
MOVL C02077 V=800.0 PL=0
MOVL C02078 V=800.0 PL=0
MOVL C02079 V=800.0 PL=0
MOVL C02080 V=800.0 PL=0
MOVL C02081 V=800.0 PL=0
MOVL C02082 V=800.0 PL=0
MOVL C02083 V=800.0 PL=0
MOVL C02084 V=800.0 PL=0
MOVL C02085 V=800.0 PL=0
MOVL C02086 V=800.0 PL=0
MOVL C02087 V=800.0 PL=0
MOVL C02088 V=800.0 PL=0
MOVL C02089 V=800.0 PL=0
MOVL C02090 V=800.0 PL=0
MOVL C02091 V=800.0 PL=0
MOVL C02092 V=800.0 PL=0
MOVL C02093 V=800.0 PL=0
MOVL C02094 V=800.0 PL=0
MOVL C02095 V=800.0 PL=0
MOVL C02096 V=800.0 PL=0
MOVL C02097 V=800.0 PL=0
MOVL C02098 V=800.0 PL=0
MOVL C02099 V=800.0 PL=0
MOVL C02100 V=800.0 PL=0
MOVL C02101 V=800.0 PL=0
MOVL C02102 V=800.0 PL=0
MOVL C02103 V=800.0 PL=0
MOVL C02104 V=800.0 PL=0
MOVL C02105 V=800.0 PL=0
MOVL C02106 V=800.0 PL=0
MOVL C02107 V=800.0 PL=0
MOVL C02108 V=800.0 PL=0
MOVL C02109 V=800.0 PL=0
MOVL C02110 V=800.0 PL=0
MOVL C02111 V=800.0 PL=0
MOVL C02112 V=800.0 PL=0
MOVL C02113 V=800.0 PL=0
MOVL C02114 V=800.0 PL=0
MOVL C02115 V=800.0 PL=0
MOVL C02116 V=800.0 PL=0
MOVL C02117 V=800.0 PL=0
MOVL C02118 V=800.0 PL=0
MOVL C02119 V=800.0 PL=0
MOVL C02120 V=800.0 PL=0
MOVL C02121 V=800.0 PL=0
MOVL C02122 V=800.0 PL=0
MOVL C02123 V=800.0 PL=0
MOVL C02124 V=800.0 PL=0
MOVL C02125 V=800.0 PL=0
MOVL C02126 V=800.0 PL=0
MOVL C02127 V=800.0 PL=0
MOVL C02128 V=800.0 PL=0
MOVL C02129 V=800.0 PL=0
MOVL C02130 V=800.0 PL=0
MOVL C02131 V=800.0 PL=0
MOVL C02132 V=800.0 PL=0
MOVL C02133 V=800.0 PL=0
MOVL C02134 V=800.0 PL=0
MOVL C02135 V=800.0 PL=0
MOVL C02136 V=800.0 PL=0
MOVL C02137 V=800.0 PL=0
MOVL C02138 V=800.0 PL=0
MOVL C02139 V=800.0 PL=0
MOVL C02140 V=800.0 PL=0
MOVL C02141 V=800.0 PL=0
MOVL C02142 V=800.0 PL=0
MOVL C02143 V=800.0 PL=0
MOVL C02144 V=800.0 PL=0
MOVL C02145 V=800.0 PL=0
MOVL C02146 V=800.0 PL=0
MOVL C02147 V=800.0 PL=0
MOVL C02148 V=800.0 PL=0
MOVL C02149 V=800.0 PL=0
MOVL C02150 V=800.0 PL=0
MOVL C02151 V=800.0 PL=0
MOVL C02152 V=800.0 PL=0
MOVL C02153 V=800.0 PL=0
MOVL C02154 V=800.0 PL=0
MOVL C02155 V=800.0 PL=0
MOVL C02156 V=800.0 PL=0
MOVL C02157 V=800.0 PL=0
MOVL C02158 V=800.0 PL=0
MOVL C02159 V=800.0 PL=0
MOVL C02160 V=800.0 PL=0
MOVL C02161 V=800.0 PL=0
MOVL C02162 V=800.0 PL=0
MOVL C02163 V=800.0 PL=0
MOVL C02164 V=800.0 PL=0
MOVL C02165 V=800.0 PL=0
MOVL C02166 V=800.0 PL=0
MOVL C02167 V=800.0 PL=0
MOVL C02168 V=800.0 PL=0
MOVL C02169 V=800.0 PL=0
MOVL C02170 V=800.0 PL=0
MOVL C02171 V=800.0 PL=0
MOVL C02172 V=800.0 PL=0
MOVL C02173 V=800.0 PL=0
MOVL C02174 V=800.0 PL=0
MOVL C02175 V=800.0 PL=0
MOVL C02176 V=800.0 PL=0
MOVL C02177 V=800.0 PL=0
MOVL C02178 V=800.0 PL=0
MOVL C02179 V=800.0 PL=0
MOVL C02180 V=800.0 PL=0
MOVL C02181 V=800.0 PL=0
MOVL C02182 V=800.0 PL=0
MOVL C02183 V=800.0 PL=0
MOVL C02184 V=800.0 PL=0
MOVL C02185 V=800.0 PL=0
MOVL C02186 V=800.0 PL=0
MOVL C02187 V=800.0 PL=0
MOVL C02188 V=800.0 PL=0
MOVL C02189 V=800.0 PL=0
MOVL C02190 V=800.0 PL=0
MOVL C02191 V=800.0 PL=0
MOVL C02192 V=800.0 PL=0
MOVL C02193 V=800.0 PL=0
MOVL C02194 V=800.0 PL=0
MOVL C02195 V=800.0 PL=0
MOVL C02196 V=800.0 PL=0
MOVL C02197 V=800.0 PL=0
MOVL C02198 V=800.0 PL=0
MOVL C02199 V=800.0 PL=0
MOVL C02200 V=800.0 PL=0
MOVL C02201 V=800.0 PL=0
MOVL C02202 V=800.0 PL=0
MOVL C02203 V=800.0 PL=0
MOVL C02204 V=800.0 PL=0
MOVL C02205 V=800.0 PL=0
MOVL C02206 V=800.0 PL=0
MOVL C02207 V=800.0 PL=0
MOVL C02208 V=800.0 PL=0
MOVL C02209 V=800.0 PL=0
MOVL C02210 V=800.0 PL=0
MOVL C02211 V=800.0 PL=0
MOVL C02212 V=800.0 PL=0
MOVL C02213 V=800.0 PL=0
MOVL C02214 V=800.0 PL=0
MOVL C02215 V=800.0 PL=0
MOVL C02216 V=800.0 PL=0
MOVL C02217 V=800.0 PL=0
MOVL C02218 V=800.0 PL=0
MOVL C02219 V=800.0 PL=0
MOVL C02220 V=800.0 PL=0
MOVL C02221 V=800.0 PL=0
MOVL C02222 V=800.0 PL=0
MOVL C02223 V=800.0 PL=0
MOVL C02224 V=800.0 PL=0
MOVL C02225 V=800.0 PL=0
MOVL C02226 V=800.0 PL=0
MOVL C02227 V=800.0 PL=0
MOVL C02228 V=800.0 PL=0
MOVL C02229 V=800.0 PL=0
MOVL C02230 V=800.0 PL=0
MOVL C02231 V=800.0 PL=0
MOVL C02232 V=800.0 PL=0
MOVL C02233 V=800.0 PL=0
MOVL C02234 V=800.0 PL=0
MOVL C02235 V=800.0 PL=0
MOVL C02236 V=800.0 PL=0
MOVL C02237 V=800.0 PL=0
MOVL C02238 V=800.0 PL=0
MOVL C02239 V=800.0 PL=0
MOVL C02240 V=800.0 PL=0
MOVL C02241 V=800.0 PL=0
MOVL C02242 V=800.0 PL=0
MOVL C02243 V=800.0 PL=0
MOVL C02244 V=800.0 PL=0
MOVL C02245 V=800.0 PL=0
MOVL C02246 V=800.0 PL=0
MOVL C02247 V=800.0 PL=0
MOVL C02248 V=800.0 PL=0
MOVL C02249 V=800.0 PL=0
MOVL C02250 V=800.0 PL=0
MOVL C02251 V=800.0 PL=0
MOVL C02252 V=800.0 PL=0
MOVL C02253 V=800.0 PL=0
MOVL C02254 V=800.0 PL=0
MOVL C02255 V=800.0 PL=0
MOVL C02256 V=800.0 PL=0
MOVL C02257 V=800.0 PL=0
MOVL C02258 V=800.0 PL=0
MOVL C02259 V=800.0 PL=0
MOVL C02260 V=800.0 PL=0
MOVL C02261 V=800.0 PL=0
MOVL C02262 V=800.0 PL=0
MOVL C02263 V=800.0 PL=0
MOVL C02264 V=800.0 PL=0
MOVL C02265 V=800.0 PL=0
MOVL C02266 V=800.0 PL=0
MOVL C02267 V=800.0 PL=0
MOVL C02268 V=800.0 PL=0
MOVL C02269 V=800.0 PL=0
MOVL C02270 V=800.0 PL=0
MOVL C02271 V=800.0 PL=0
MOVL C02272 V=800.0 PL=0
MOVL C02273 V=800.0 PL=0
MOVL C02274 V=800.0 PL=0
MOVL C02275 V=800.0 PL=0
MOVL C02276 V=800.0 PL=0
MOVL C02277 V=800.0 PL=0
MOVL C02278 V=800.0 PL=0
MOVL C02279 V=800.0 PL=0
MOVL C02280 V=800.0 PL=0
MOVL C02281 V=800.0 PL=0
MOVL C02282 V=800.0 PL=0
MOVL C02283 V=800.0 PL=0
MOVL C02284 V=800.0 PL=0
MOVL C02285 V=800.0 PL=0
MOVL C02286 V=800.0 PL=0
MOVL C02287 V=800.0 PL=0
MOVL C02288 V=800.0 PL=0
MOVL C02289 V=800.0 PL=0
MOVL C02290 V=800.0 PL=0
MOVL C02291 V=800.0 PL=0
MOVL C02292 V=800.0 PL=0
MOVL C02293 V=800.0 PL=0
MOVL C02294 V=800.0 PL=0
MOVL C02295 V=800.0 PL=0
MOVL C02296 V=800.0 PL=0
MOVL C02297 V=800.0 PL=0
MOVL C02298 V=800.0 PL=0
MOVL C02299 V=800.0 PL=0
MOVL C02300 V=800.0 PL=0
MOVL C02301 V=800.0 PL=0
MOVL C02302 V=800.0 PL=0
MOVL C02303 V=800.0 PL=0
MOVL C02304 V=800.0 PL=0
MOVL C02305 V=800.0 PL=0
MOVL C02306 V=800.0 PL=0
MOVL C02307 V=800.0 PL=0
MOVL C02308 V=800.0 PL=0
MOVL C02309 V=800.0 PL=0
MOVL C02310 V=800.0 PL=0
MOVL C02311 V=800.0 PL=0
MOVL C02312 V=800.0 PL=0
MOVL C02313 V=800.0 PL=0
MOVL C02314 V=800.0 PL=0
MOVL C02315 V=800.0 PL=0
MOVL C02316 V=800.0 PL=0
MOVL C02317 V=800.0 PL=0
MOVL C02318 V=800.0 PL=0
MOVL C02319 V=800.0 PL=0
MOVL C02320 V=800.0 PL=0
MOVL C02321 V=800.0 PL=0
MOVL C02322 V=800.0 PL=0
MOVL C02323 V=800.0 PL=0
MOVL C02324 V=800.0 PL=0
MOVL C02325 V=800.0 PL=0
MOVL C02326 V=800.0 PL=0
MOVL C02327 V=800.0 PL=0
MOVL C02328 V=800.0 PL=0
MOVL C02329 V=800.0 PL=0
MOVL C02330 V=800.0 PL=0
MOVL C02331 V=800.0 PL=0
MOVL C02332 V=800.0 PL=0
MOVL C02333 V=800.0 PL=0
MOVL C02334 V=800.0 PL=0
MOVL C02335 V=800.0 PL=0
MOVL C02336 V=800.0 PL=0
MOVL C02337 V=800.0 PL=0
MOVL C02338 V=800.0 PL=0
MOVL C02339 V=800.0 PL=0
MOVL C02340 V=800.0 PL=0
MOVL C02341 V=800.0 PL=0
MOVL C02342 V=800.0 PL=0
MOVL C02343 V=800.0 PL=0
MOVL C02344 V=800.0 PL=0
MOVL C02345 V=800.0 PL=0
MOVL C02346 V=800.0 PL=0
MOVL C02347 V=800.0 PL=0
MOVL C02348 V=800.0 PL=0
MOVL C02349 V=800.0 PL=0
MOVL C02350 V=800.0 PL=0
MOVL C02351 V=800.0 PL=0
MOVL C02352 V=800.0 PL=0
MOVL C02353 V=800.0 PL=0
MOVL C02354 V=800.0 PL=0
MOVL C02355 V=800.0 PL=0
MOVL C02356 V=800.0 PL=0
MOVL C02357 V=800.0 PL=0
MOVL C02358 V=800.0 PL=0
MOVL C02359 V=800.0 PL=0
MOVL C02360 V=800.0 PL=0
MOVL C02361 V=800.0 PL=0
MOVL C02362 V=800.0 PL=0
MOVL C02363 V=800.0 PL=0
MOVL C02364 V=800.0 PL=0
MOVL C02365 V=800.0 PL=0
MOVL C02366 V=800.0 PL=0
MOVL C02367 V=800.0 PL=0
MOVL C02368 V=800.0 PL=0
MOVL C02369 V=800.0 PL=0
MOVL C02370 V=800.0 PL=0
MOVL C02371 V=800.0 PL=0
MOVL C02372 V=800.0 PL=0
MOVL C02373 V=800.0 PL=0
MOVL C02374 V=800.0 PL=0
MOVL C02375 V=800.0 PL=0
MOVL C02376 V=800.0 PL=0
MOVL C02377 V=800.0 PL=0
MOVL C02378 V=800.0 PL=0
MOVL C02379 V=800.0 PL=0
MOVL C02380 V=800.0 PL=0
MOVL C02381 V=800.0 PL=0
MOVL C02382 V=800.0 PL=0
MOVL C02383 V=800.0 PL=0
MOVL C02384 V=800.0 PL=0
MOVL C02385 V=800.0 PL=0
MOVL C02386 V=800.0 PL=0
MOVL C02387 V=800.0 PL=0
MOVL C02388 V=800.0 PL=0
MOVL C02389 V=800.0 PL=0
MOVL C02390 V=800.0 PL=0
MOVL C02391 V=800.0 PL=0
MOVL C02392 V=800.0 PL=0
MOVL C02393 V=800.0 PL=0
MOVL C02394 V=800.0 PL=0
MOVL C02395 V=800.0 PL=0
MOVL C02396 V=800.0 PL=0
MOVL C02397 V=800.0 PL=0
MOVL C02398 V=800.0 PL=0
MOVL C02399 V=800.0 PL=0
MOVL C02400 V=800.0 PL=0
MOVL C02401 V=800.0 PL=0
MOVL C02402 V=800.0 PL=0
MOVL C02403 V=800.0 PL=0
MOVL C02404 V=800.0 PL=0
MOVL C02405 V=800.0 PL=0
MOVL C02406 V=800.0 PL=0
MOVL C02407 V=800.0 PL=0
MOVL C02408 V=800.0 PL=0
MOVL C02409 V=800.0 PL=0
MOVL C02410 V=800.0 PL=0
MOVL C02411 V=800.0 PL=0
MOVL C02412 V=800.0 PL=0
MOVL C02413 V=800.0 PL=0
MOVL C02414 V=800.0 PL=0
MOVL C02415 V=800.0 PL=0
MOVL C02416 V=800.0 PL=0
MOVL C02417 V=800.0 PL=0
MOVL C02418 V=800.0 PL=0
MOVL C02419 V=800.0 PL=0
MOVL C02420 V=800.0 PL=0
MOVL C02421 V=800.0 PL=0
MOVL C02422 V=800.0 PL=0
MOVL C02423 V=800.0 PL=0
MOVL C02424 V=800.0 PL=0
MOVL C02425 V=800.0 PL=0
MOVL C02426 V=800.0 PL=0
MOVL C02427 V=800.0 PL=0
MOVL C02428 V=800.0 PL=0
MOVL C02429 V=800.0 PL=0
MOVL C02430 V=800.0 PL=0
MOVL C02431 V=800.0 PL=0
